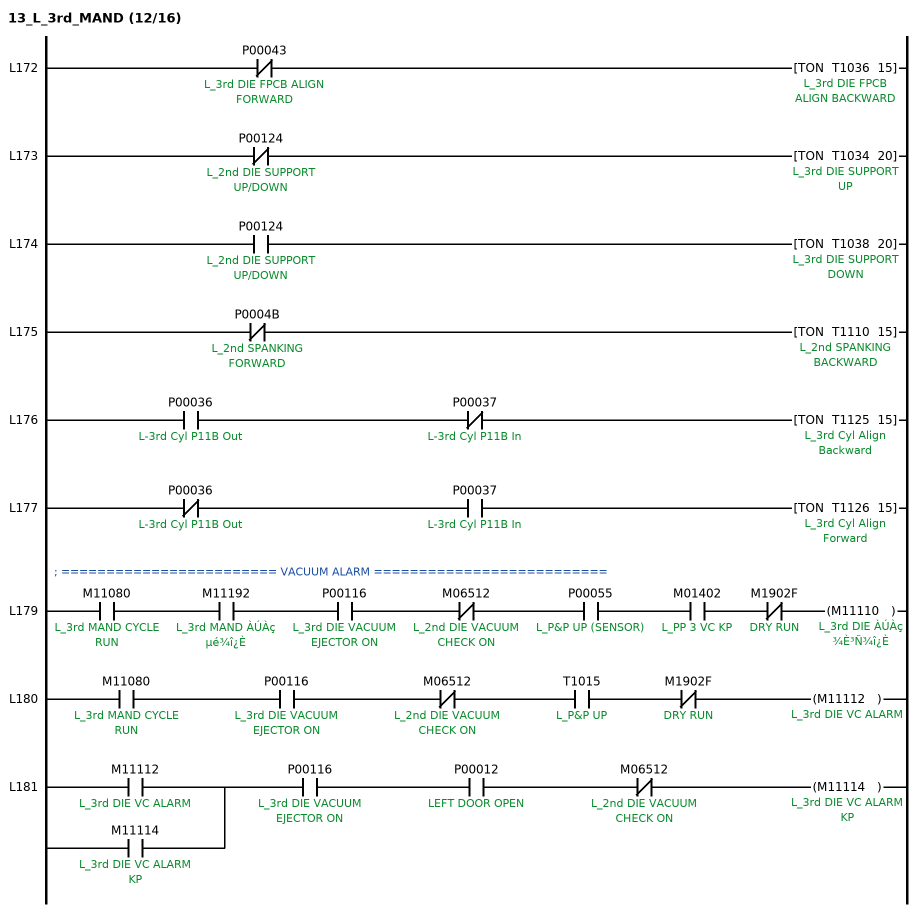
[picture p96: 13_L_3rd_MAND rungs L172-L181]
; L172
LOAD NOT  P00043	// L_3rd DIE FPCB ALIGN FORWARD
TON       T1036 15	// L_3rd DIE FPCB ALIGN BACKWARD
; L173
LOAD NOT  P00124	// L_2nd DIE SUPPORT UP/DOWN
TON       T1034 20	// L_3rd DIE SUPPORT UP
; L174
LOAD      P00124	// L_2nd DIE SUPPORT UP/DOWN
TON       T1038 20	// L_3rd DIE SUPPORT DOWN
; L175
LOAD NOT  P0004B	// L_2nd SPANKING FORWARD
TON       T1110 15	// L_2nd SPANKING BACKWARD
; L176
LOAD      P00036	// L-3rd Cyl P11B Out
AND NOT   P00037	// L-3rd Cyl P11B In
TON       T1125 15	// L_3rd Cyl Align Backward
; L177
LOAD NOT  P00036	// L-3rd Cyl P11B Out
AND       P00037	// L-3rd Cyl P11B In
TON       T1126 15	// L_3rd Cyl Align Forward
// ======================== VACUUM ALARM ==========================
; L179
LOAD      M11080	// L_3rd MAND CYCLE RUN
AND       M11192	// L_3rd MAND ÀÚÀç µé¾î¿È
AND       P00116	// L_3rd DIE VACUUM EJECTOR ON
AND NOT   M06512	// L_2nd DIE VACUUM CHECK ON
AND       P00055	// L_P&P UP (SENSOR)
AND       M01402	// L_PP 3 VC KP
AND NOT   M1902F	// DRY RUN
OUT       M11110	// L_3rd DIE ÀÚÀç ¾È³Ñ¾î¿È
; L180
LOAD      M11080	// L_3rd MAND CYCLE RUN
AND       P00116	// L_3rd DIE VACUUM EJECTOR ON
AND NOT   M06512	// L_2nd DIE VACUUM CHECK ON
AND       T1015	// L_P&P UP
AND NOT   M1902F	// DRY RUN
OUT       M11112	// L_3rd DIE VC ALARM
; L181
LOAD      M11112	// L_3rd DIE VC ALARM
OR        M11114	// L_3rd DIE VC ALARM KP
AND       P00116	// L_3rd DIE VACUUM EJECTOR ON
AND       P00012	// LEFT DOOR OPEN
AND NOT   M06512	// L_2nd DIE VACUUM CHECK ON
OUT       M11114	// L_3rd DIE VC ALARM KP

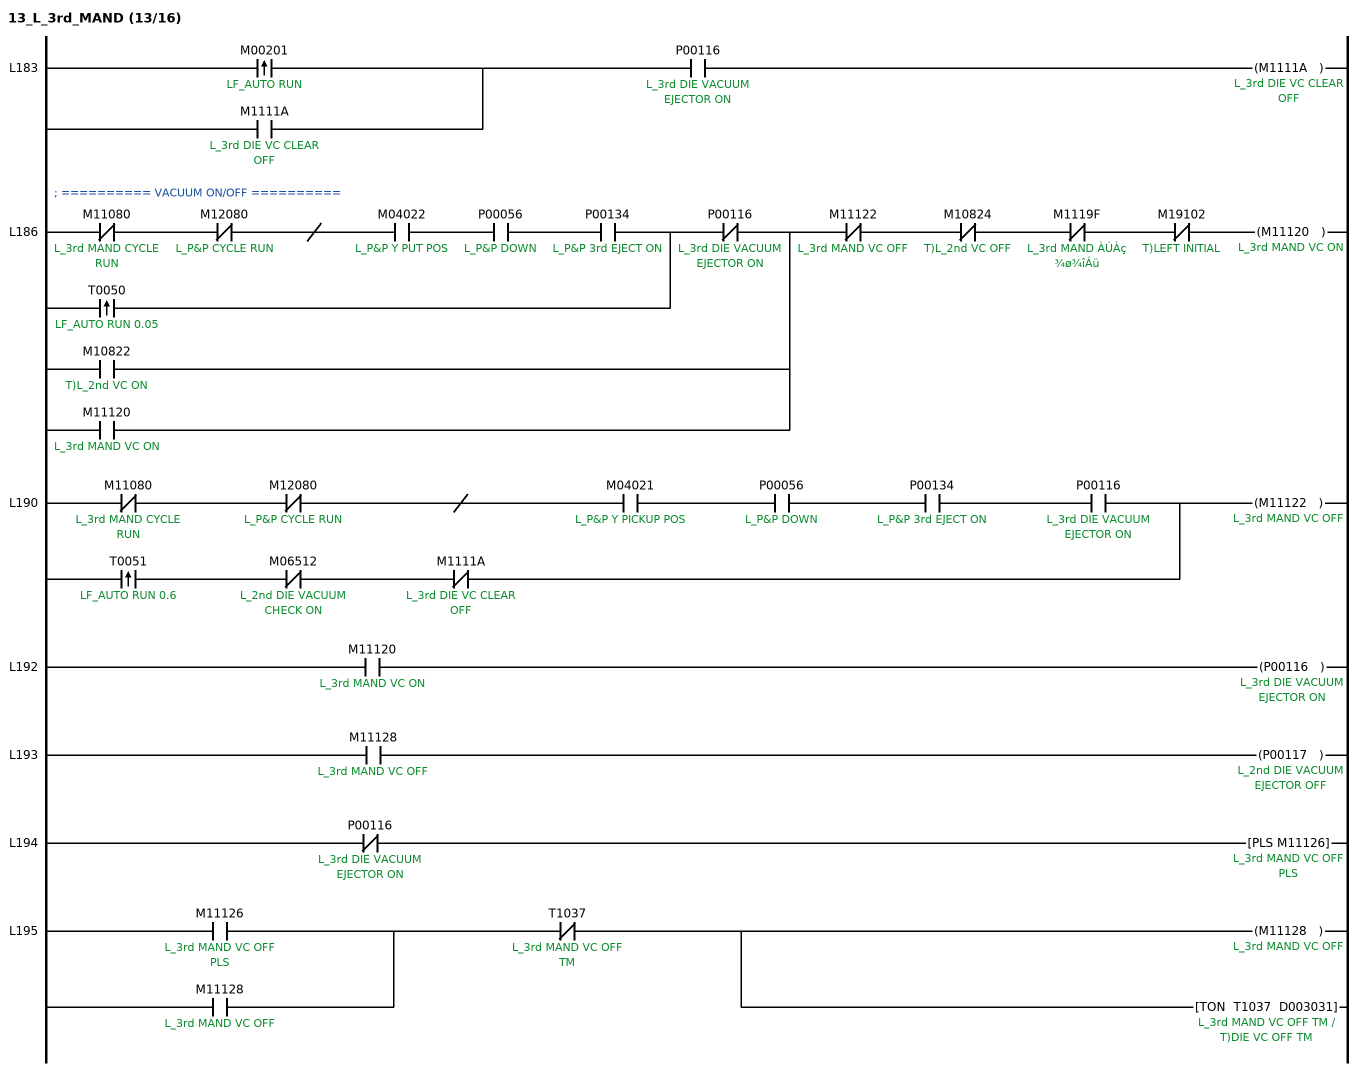
; L183
LOADP     M00201	// LF_AUTO RUN
OR        M1111A	// L_3rd DIE VC CLEAR OFF
AND       P00116	// L_3rd DIE VACUUM EJECTOR ON
OUT       M1111A	// L_3rd DIE VC CLEAR OFF
// ========== VACUUM ON/OFF ==========
; L186
LOAD NOT  M11080	// L_3rd MAND CYCLE RUN
AND NOT   M12080	// L_P&P CYCLE RUN
NOT
AND       M04022	// L_P&P Y PUT POS
AND       P00056	// L_P&P DOWN
AND       P00134	// L_P&P 3rd EJECT ON
ORP       T0050	// LF_AUTO RUN 0.05
AND NOT   P00116	// L_3rd DIE VACUUM EJECTOR ON
OR        M10822	// T)L_2nd VC ON
OR        M11120	// L_3rd MAND VC ON
AND NOT   M11122	// L_3rd MAND VC OFF
AND NOT   M10824	// T)L_2nd VC OFF
AND NOT   M1119F	// L_3rd MAND ÀÚÀç ¾ø¾îÁü
AND NOT   M19102	// T)LEFT INITIAL
OUT       M11120	// L_3rd MAND VC ON
; L190
LOAD NOT  M11080	// L_3rd MAND CYCLE RUN
AND NOT   M12080	// L_P&P CYCLE RUN
NOT
AND       M04021	// L_P&P Y PICKUP POS
AND       P00056	// L_P&P DOWN
AND       P00134	// L_P&P 3rd EJECT ON
AND       P00116	// L_3rd DIE VACUUM EJECTOR ON
LOADP     T0051	// LF_AUTO RUN 0.6
AND NOT   M06512	// L_2nd DIE VACUUM CHECK ON
AND NOT   M1111A	// L_3rd DIE VC CLEAR OFF
OR LOAD
OUT       M11122	// L_3rd MAND VC OFF
; L192
LOAD      M11120	// L_3rd MAND VC ON
OUT       P00116	// L_3rd DIE VACUUM EJECTOR ON
; L193
LOAD      M11128	// L_3rd MAND VC OFF
OUT       P00117	// L_2nd DIE VACUUM EJECTOR OFF
; L194
LOAD NOT  P00116	// L_3rd DIE VACUUM EJECTOR ON
OUTP      M11126	// L_3rd MAND VC OFF PLS
; L195
LOAD      M11126	// L_3rd MAND VC OFF PLS
OR        M11128	// L_3rd MAND VC OFF
AND NOT   T1037	// L_3rd MAND VC OFF TM
OUT       M11128	// L_3rd MAND VC OFF
TON       T1037 D003031	// L_3rd MAND VC OFF TM / T)DIE VC OFF TM

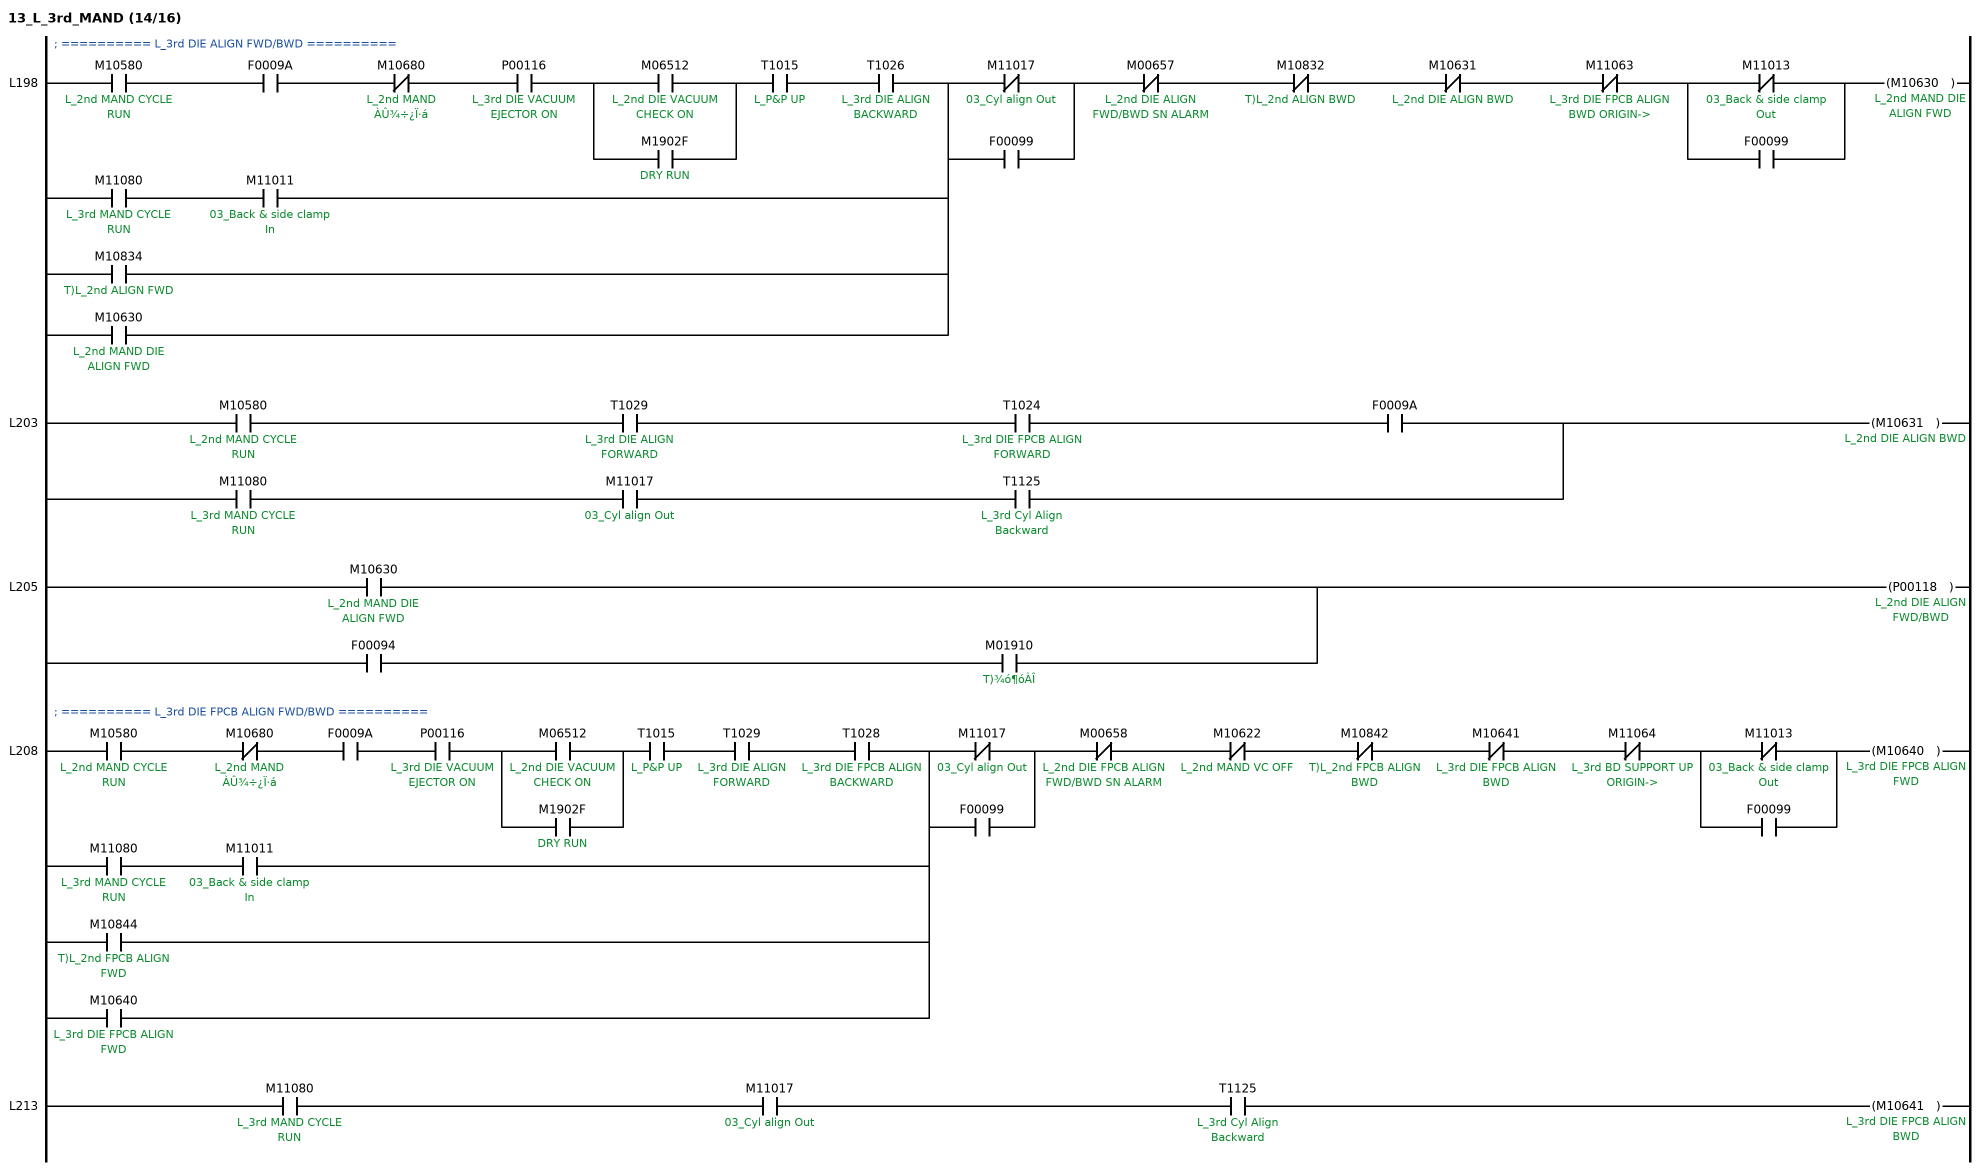
// ========== L_3rd DIE ALIGN FWD/BWD ==========
; L198
LOAD      M10580	// L_2nd MAND CYCLE RUN
AND       F0009A
AND NOT   M10680	// L_2nd MAND ÀÛ¾÷¿Ï·á
AND       P00116	// L_3rd DIE VACUUM EJECTOR ON
LOAD      M06512	// L_2nd DIE VACUUM CHECK ON
OR        M1902F	// DRY RUN
AND LOAD
AND       T1015	// L_P&P UP
AND       T1026	// L_3rd DIE ALIGN BACKWARD
LOAD      M11080	// L_3rd MAND CYCLE RUN
AND       M11011	// 03_Back & side clamp In
OR LOAD
OR        M10834	// T)L_2nd ALIGN FWD
OR        M10630	// L_2nd MAND DIE ALIGN FWD
LOAD NOT  M11017	// 03_Cyl align Out
OR        F00099
AND LOAD
AND NOT   M00657	// L_2nd DIE ALIGN FWD/BWD SN ALARM
AND NOT   M10832	// T)L_2nd ALIGN BWD
AND NOT   M10631	// L_2nd DIE ALIGN BWD
AND NOT   M11063	// L_3rd DIE FPCB ALIGN BWD ORIGIN->
LOAD NOT  M11013	// 03_Back & side clamp Out
OR        F00099
AND LOAD
OUT       M10630	// L_2nd MAND DIE ALIGN FWD
; L203
LOAD      M10580	// L_2nd MAND CYCLE RUN
AND       T1029	// L_3rd DIE ALIGN FORWARD
AND       T1024	// L_3rd DIE FPCB ALIGN FORWARD
AND       F0009A
LOAD      M11080	// L_3rd MAND CYCLE RUN
AND       M11017	// 03_Cyl align Out
AND       T1125	// L_3rd Cyl Align Backward
OR LOAD
OUT       M10631	// L_2nd DIE ALIGN BWD
; L205
LOAD      M10630	// L_2nd MAND DIE ALIGN FWD
LOAD      F00094
AND       M01910	// T)¾ó¶óÀÎ
OR LOAD
OUT       P00118	// L_2nd DIE ALIGN FWD/BWD
// ========== L_3rd DIE FPCB ALIGN FWD/BWD ==========
; L208
LOAD      M10580	// L_2nd MAND CYCLE RUN
AND NOT   M10680	// L_2nd MAND ÀÛ¾÷¿Ï·á
AND       F0009A
AND       P00116	// L_3rd DIE VACUUM EJECTOR ON
LOAD      M06512	// L_2nd DIE VACUUM CHECK ON
OR        M1902F	// DRY RUN
AND LOAD
AND       T1015	// L_P&P UP
AND       T1029	// L_3rd DIE ALIGN FORWARD
AND       T1028	// L_3rd DIE FPCB ALIGN BACKWARD
LOAD      M11080	// L_3rd MAND CYCLE RUN
AND       M11011	// 03_Back & side clamp In
OR LOAD
OR        M10844	// T)L_2nd FPCB ALIGN FWD
OR        M10640	// L_3rd DIE FPCB ALIGN FWD
LOAD NOT  M11017	// 03_Cyl align Out
OR        F00099
AND LOAD
AND NOT   M00658	// L_2nd DIE FPCB ALIGN FWD/BWD SN ALARM
AND NOT   M10622	// L_2nd MAND VC OFF
AND NOT   M10842	// T)L_2nd FPCB ALIGN BWD
AND NOT   M10641	// L_3rd DIE FPCB ALIGN BWD
AND NOT   M11064	// L_3rd BD SUPPORT UP ORIGIN->
LOAD NOT  M11013	// 03_Back & side clamp Out
OR        F00099
AND LOAD
OUT       M10640	// L_3rd DIE FPCB ALIGN FWD
; L213
LOAD      M11080	// L_3rd MAND CYCLE RUN
AND       M11017	// 03_Cyl align Out
AND       T1125	// L_3rd Cyl Align Backward
OUT       M10641	// L_3rd DIE FPCB ALIGN BWD

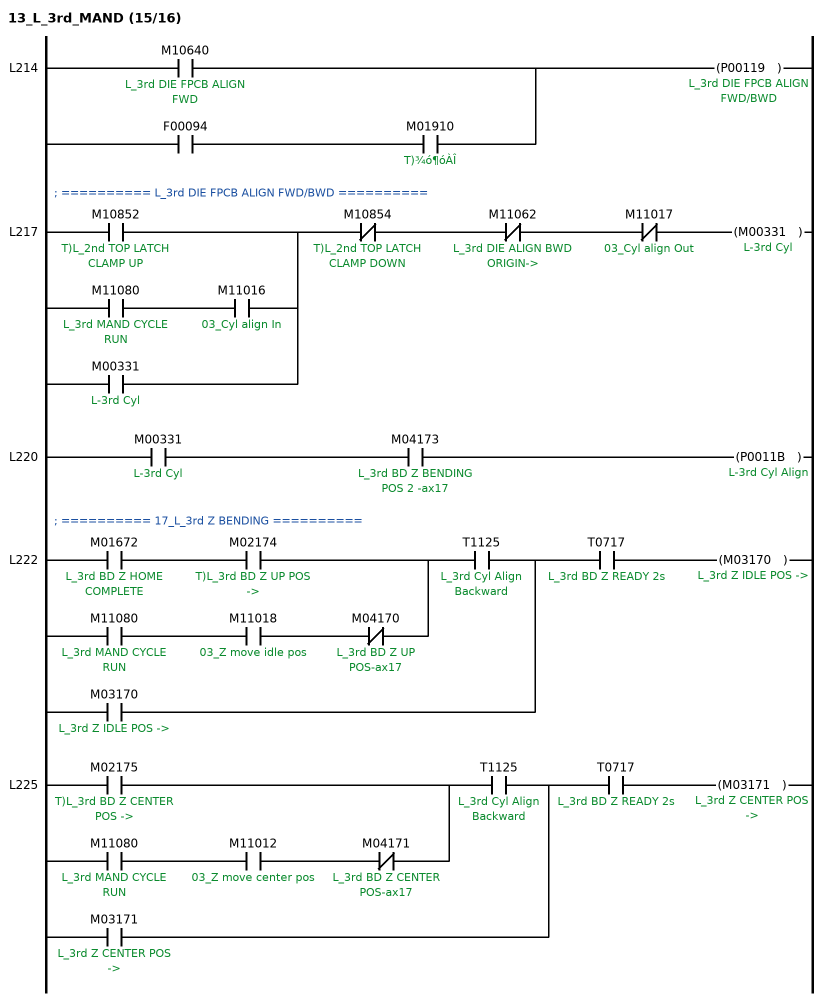
; L214
LOAD      M10640	// L_3rd DIE FPCB ALIGN FWD
LOAD      F00094
AND       M01910	// T)¾ó¶óÀÎ
OR LOAD
OUT       P00119	// L_3rd DIE FPCB ALIGN FWD/BWD
// ========== L_3rd DIE FPCB ALIGN FWD/BWD ==========
; L217
LOAD      M10852	// T)L_2nd TOP LATCH CLAMP UP
LOAD      M11080	// L_3rd MAND CYCLE RUN
AND       M11016	// 03_Cyl align In
OR LOAD
OR        M00331	// L-3rd Cyl
AND NOT   M10854	// T)L_2nd TOP LATCH CLAMP DOWN
AND NOT   M11062	// L_3rd DIE ALIGN BWD ORIGIN->
AND NOT   M11017	// 03_Cyl align Out
OUT       M00331	// L-3rd Cyl
; L220
LOAD      M00331	// L-3rd Cyl
AND       M04173	// L_3rd BD Z BENDING POS 2 -ax17
OUT       P0011B	// L-3rd Cyl Align
// ========== 17_L_3rd Z BENDING ==========
; L222
LOAD      M01672	// L_3rd BD Z HOME COMPLETE
AND       M02174	// T)L_3rd BD Z UP POS ->
LOAD      M11080	// L_3rd MAND CYCLE RUN
AND       M11018	// 03_Z move idle pos
AND NOT   M04170	// L_3rd BD Z UP POS-ax17
OR LOAD
AND       T1125	// L_3rd Cyl Align Backward
OR        M03170	// L_3rd Z IDLE POS ->
AND       T0717	// L_3rd BD Z READY 2s
OUT       M03170	// L_3rd Z IDLE POS ->
; L225
LOAD      M02175	// T)L_3rd BD Z CENTER POS ->
LOAD      M11080	// L_3rd MAND CYCLE RUN
AND       M11012	// 03_Z move center pos
AND NOT   M04171	// L_3rd BD Z CENTER POS-ax17
OR LOAD
AND       T1125	// L_3rd Cyl Align Backward
OR        M03171	// L_3rd Z CENTER POS ->
AND       T0717	// L_3rd BD Z READY 2s
OUT       M03171	// L_3rd Z CENTER POS ->

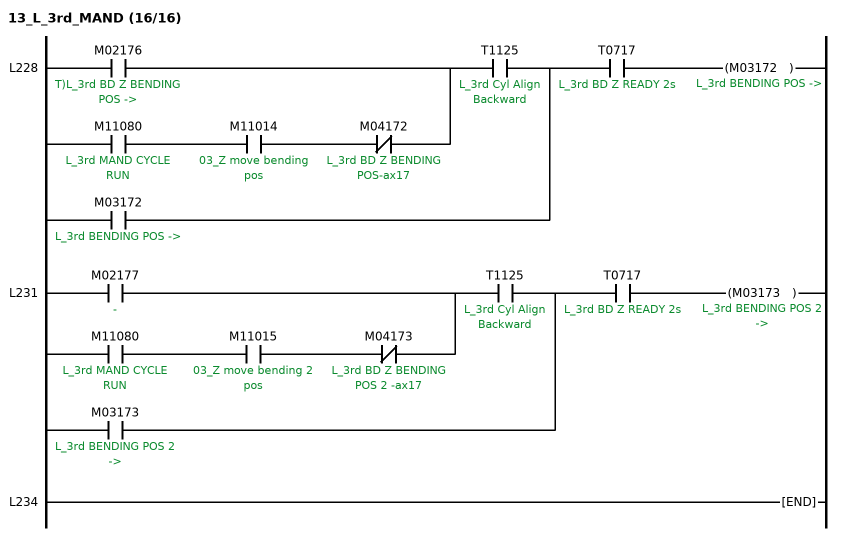
; L228
LOAD      M02176	// T)L_3rd BD Z BENDING POS ->
LOAD      M11080	// L_3rd MAND CYCLE RUN
AND       M11014	// 03_Z move bending pos
AND NOT   M04172	// L_3rd BD Z BENDING POS-ax17
OR LOAD
AND       T1125	// L_3rd Cyl Align Backward
OR        M03172	// L_3rd BENDING POS ->
AND       T0717	// L_3rd BD Z READY 2s
OUT       M03172	// L_3rd BENDING POS ->
; L231
LOAD      M02177	// -
LOAD      M11080	// L_3rd MAND CYCLE RUN
AND       M11015	// 03_Z move bending 2 pos
AND NOT   M04173	// L_3rd BD Z BENDING POS 2 -ax17
OR LOAD
AND       T1125	// L_3rd Cyl Align Backward
OR        M03173	// L_3rd BENDING POS 2 ->
AND       T0717	// L_3rd BD Z READY 2s
OUT       M03173	// L_3rd BENDING POS 2 ->
; L234
END

PROGRAM 14_L_TOOL (task: ½ºÄµ ÇÁ·Î±×·¥)

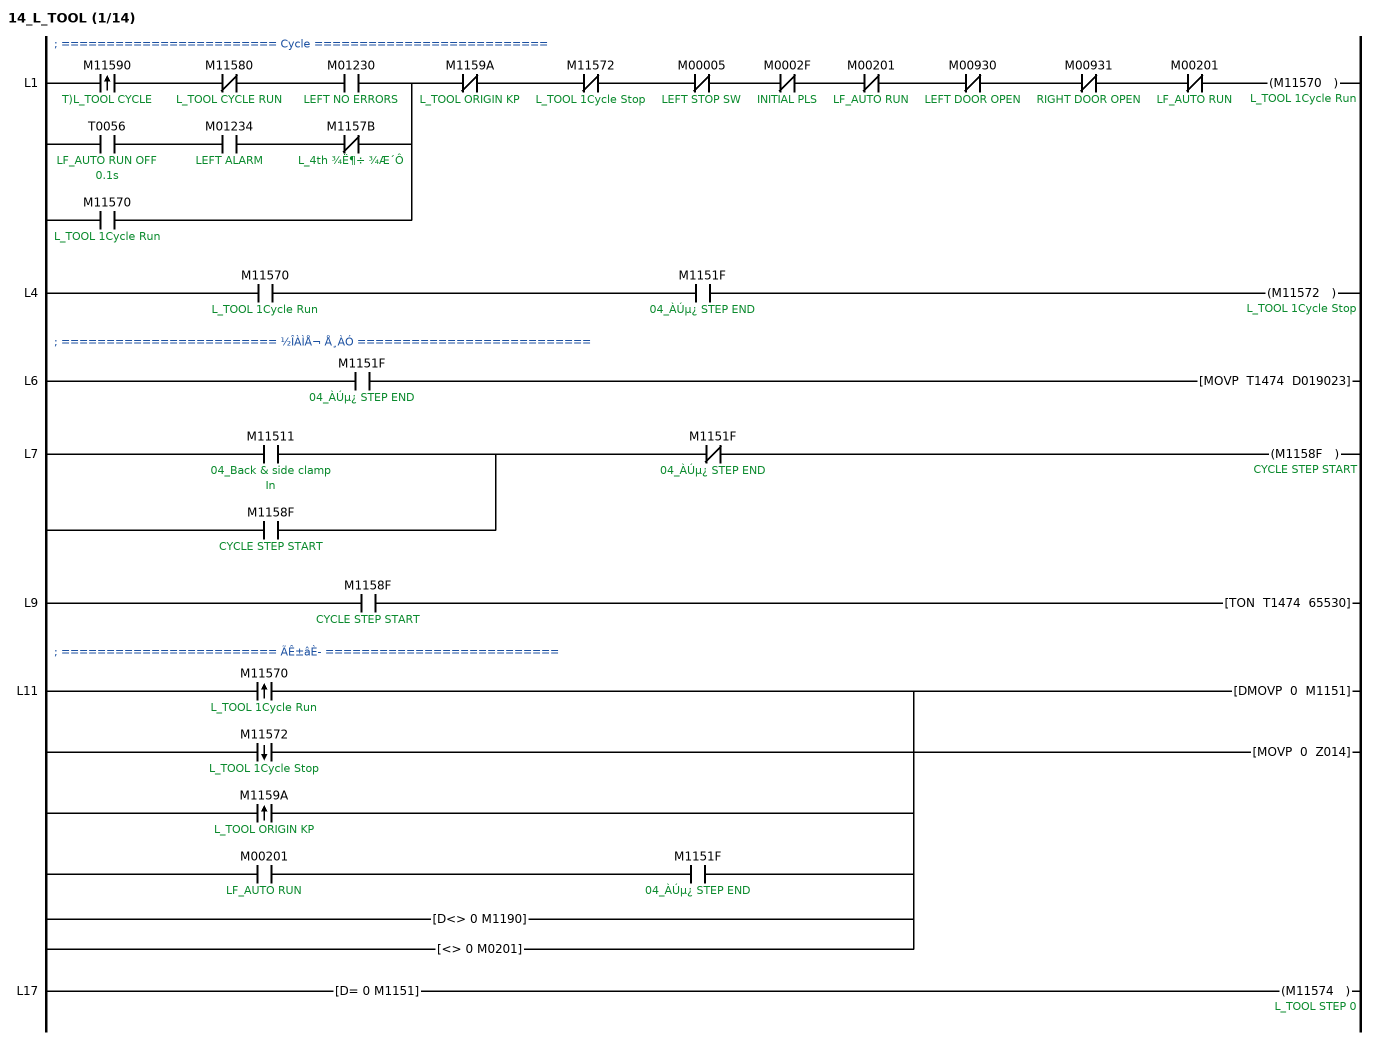
// ======================== Cycle ==========================
; L1
LOADP     M11590	// T)L_TOOL CYCLE
AND NOT   M11580	// L_TOOL CYCLE RUN
AND       M01230	// LEFT NO ERRORS
LOAD      T0056	// LF_AUTO RUN OFF 0.1s
AND       M01234	// LEFT ALARM
AND NOT   M1157B	// L_4th ¾Ë¶÷ ¾Æ´Ô
OR LOAD
OR        M11570	// L_TOOL 1Cycle Run
AND NOT   M1159A	// L_TOOL ORIGIN KP
AND NOT   M11572	// L_TOOL 1Cycle Stop
AND NOT   M00005	// LEFT STOP SW
AND NOT   M0002F	// INITIAL PLS
AND NOT   M00201	// LF_AUTO RUN
AND NOT   M00930	// LEFT DOOR OPEN
AND NOT   M00931	// RIGHT DOOR OPEN
AND NOT   M00201	// LF_AUTO RUN
OUT       M11570	// L_TOOL 1Cycle Run
; L4
LOAD      M11570	// L_TOOL 1Cycle Run
AND       M1151F	// 04_ÀÚµ¿ STEP END
OUT       M11572	// L_TOOL 1Cycle Stop
// ======================== ½ÎÀÌÅ¬ Å¸ÀÓ ==========================
; L6
LOAD      M1151F	// 04_ÀÚµ¿ STEP END
MOVP      T1474 D019023
; L7
LOAD      M11511	// 04_Back & side clamp In
OR        M1158F	// CYCLE STEP START
AND NOT   M1151F	// 04_ÀÚµ¿ STEP END
OUT       M1158F	// CYCLE STEP START
; L9
LOAD      M1158F	// CYCLE STEP START
TON       T1474 65530
// ======================== ÃÊ±âÈ­ ==========================
; L11
LOADP     M11570	// L_TOOL 1Cycle Run
ORN       M11572	// L_TOOL 1Cycle Stop
ORP       M1159A	// L_TOOL ORIGIN KP
LOAD      M00201	// LF_AUTO RUN
AND       M1151F	// 04_ÀÚµ¿ STEP END
OR LOAD
ORD<>     0 M1190
OR<>      0 M0201
DMOVP     0 M1151
MOVP      0 Z014
; L17
LOADD=    0 M1151
OUT       M11574	// L_TOOL STEP 0

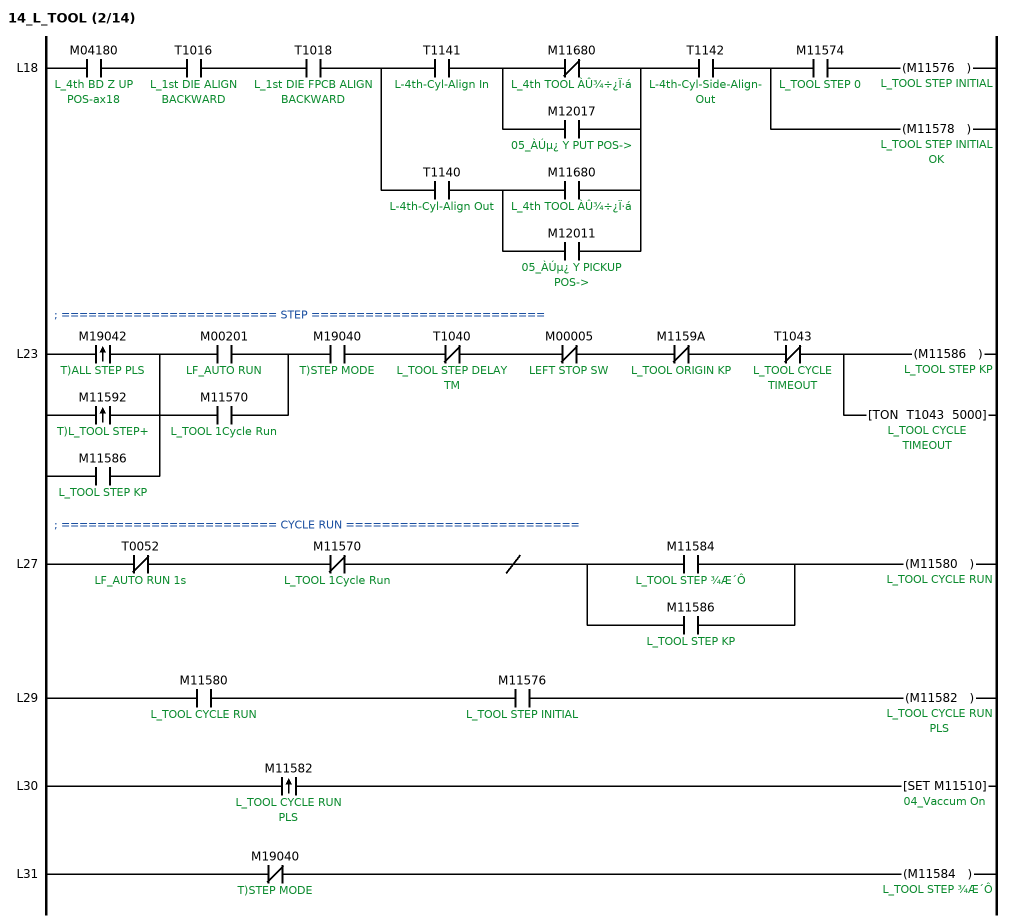
; L18
LOAD      M04180	// L_4th BD Z UP POS-ax18
AND       T1016	// L_1st DIE ALIGN BACKWARD
AND       T1018	// L_1st DIE FPCB ALIGN BACKWARD
LOAD      T1141	// L-4th-Cyl-Align In
LOAD NOT  M11680	// L_4th TOOL ÀÛ¾÷¿Ï·á
OR        M12017	// 05_ÀÚµ¿ Y PUT POS->
AND LOAD
LOAD      T1140	// L-4th-Cyl-Align Out
LOAD      M11680	// L_4th TOOL ÀÛ¾÷¿Ï·á
OR        M12011	// 05_ÀÚµ¿ Y PICKUP POS->
AND LOAD
OR LOAD
AND LOAD
AND       T1142	// L-4th-Cyl-Side-Align-Out
MPUSH
AND       M11574	// L_TOOL STEP 0
OUT       M11576	// L_TOOL STEP INITIAL
MPOP
OUT       M11578	// L_TOOL STEP INITIAL OK
// ======================== STEP ==========================
; L23
LOADP     M19042	// T)ALL STEP PLS
ORP       M11592	// T)L_TOOL STEP+
OR        M11586	// L_TOOL STEP KP
LOAD      M00201	// LF_AUTO RUN
OR        M11570	// L_TOOL 1Cycle Run
AND LOAD
AND       M19040	// T)STEP MODE
AND NOT   T1040	// L_TOOL STEP DELAY TM
AND NOT   M00005	// LEFT STOP SW
AND NOT   M1159A	// L_TOOL ORIGIN KP
AND NOT   T1043	// L_TOOL CYCLE TIMEOUT
OUT       M11586	// L_TOOL STEP KP
TON       T1043 5000	// L_TOOL CYCLE TIMEOUT
// ======================== CYCLE RUN ==========================
; L27
LOAD NOT  T0052	// LF_AUTO RUN 1s
AND NOT   M11570	// L_TOOL 1Cycle Run
NOT
LOAD      M11584	// L_TOOL STEP ¾Æ´Ô
OR        M11586	// L_TOOL STEP KP
AND LOAD
OUT       M11580	// L_TOOL CYCLE RUN
; L29
LOAD      M11580	// L_TOOL CYCLE RUN
AND       M11576	// L_TOOL STEP INITIAL
OUT       M11582	// L_TOOL CYCLE RUN PLS
; L30
LOADP     M11582	// L_TOOL CYCLE RUN PLS
SET       M11510	// 04_Vaccum On
; L31
LOAD NOT  M19040	// T)STEP MODE
OUT       M11584	// L_TOOL STEP ¾Æ´Ô

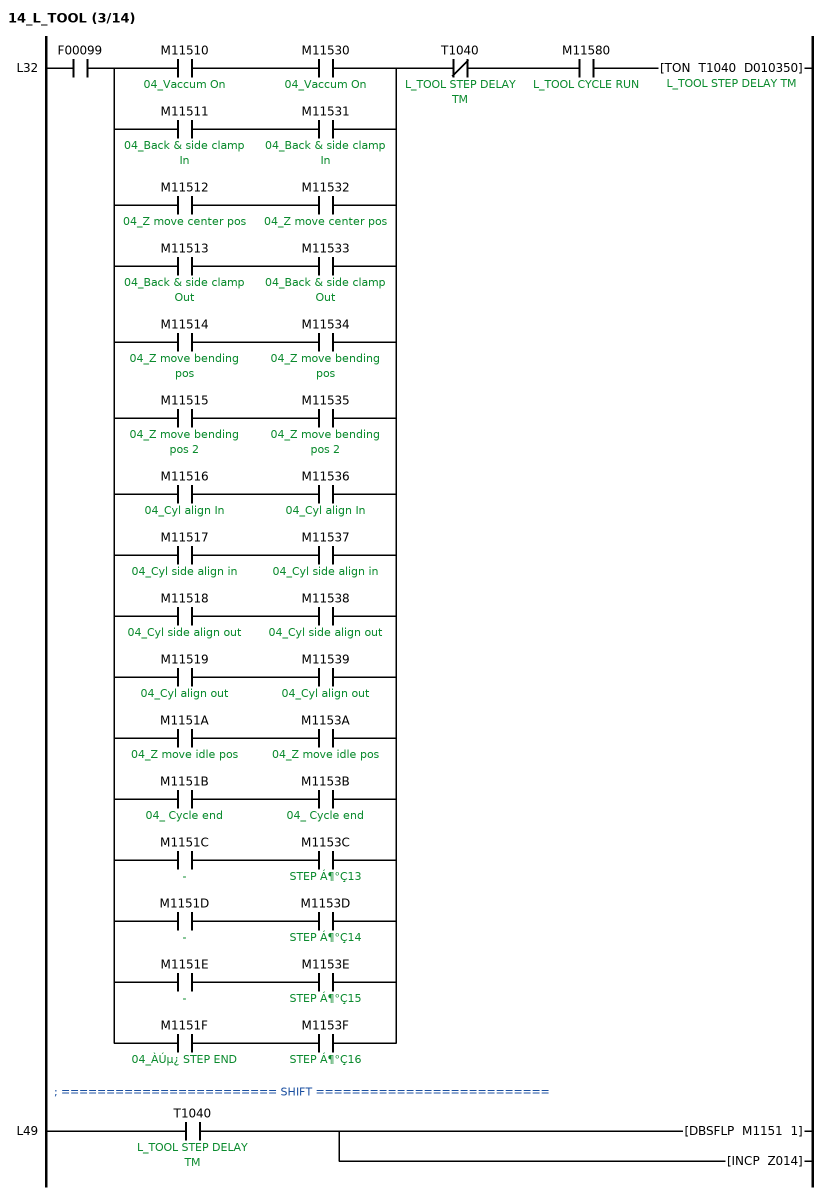
; L32
LOAD      F00099
LOAD      M11510	// 04_Vaccum On
AND       M11530	// 04_Vaccum On
LOAD      M11511	// 04_Back & side clamp In
AND       M11531	// 04_Back & side clamp In
OR LOAD
LOAD      M11512	// 04_Z move center pos
AND       M11532	// 04_Z move center pos
OR LOAD
LOAD      M11513	// 04_Back & side clamp Out
AND       M11533	// 04_Back & side clamp Out
OR LOAD
LOAD      M11514	// 04_Z move bending pos
AND       M11534	// 04_Z move bending pos
OR LOAD
LOAD      M11515	// 04_Z move bending pos 2
AND       M11535	// 04_Z move bending pos 2
OR LOAD
LOAD      M11516	// 04_Cyl align In
AND       M11536	// 04_Cyl align In
OR LOAD
LOAD      M11517	// 04_Cyl side align in
AND       M11537	// 04_Cyl side align in
OR LOAD
LOAD      M11518	// 04_Cyl side align out
AND       M11538	// 04_Cyl side align out
OR LOAD
LOAD      M11519	// 04_Cyl align out
AND       M11539	// 04_Cyl align out
OR LOAD
LOAD      M1151A	// 04_Z move idle pos
AND       M1153A	// 04_Z move idle pos
OR LOAD
LOAD      M1151B	// 04_ Cycle end
AND       M1153B	// 04_ Cycle end
OR LOAD
LOAD      M1151C	// -
AND       M1153C	// STEP Á¶°Ç13
OR LOAD
LOAD      M1151D	// -
AND       M1153D	// STEP Á¶°Ç14
OR LOAD
LOAD      M1151E	// -
AND       M1153E	// STEP Á¶°Ç15
OR LOAD
LOAD      M1151F	// 04_ÀÚµ¿ STEP END
AND       M1153F	// STEP Á¶°Ç16
OR LOAD
AND LOAD
AND NOT   T1040	// L_TOOL STEP DELAY TM
AND       M11580	// L_TOOL CYCLE RUN
TON       T1040 D010350	// L_TOOL STEP DELAY TM
// ======================== SHIFT ==========================
; L49
LOAD      T1040	// L_TOOL STEP DELAY TM
DBSFLP    M1151 1
INCP      Z014

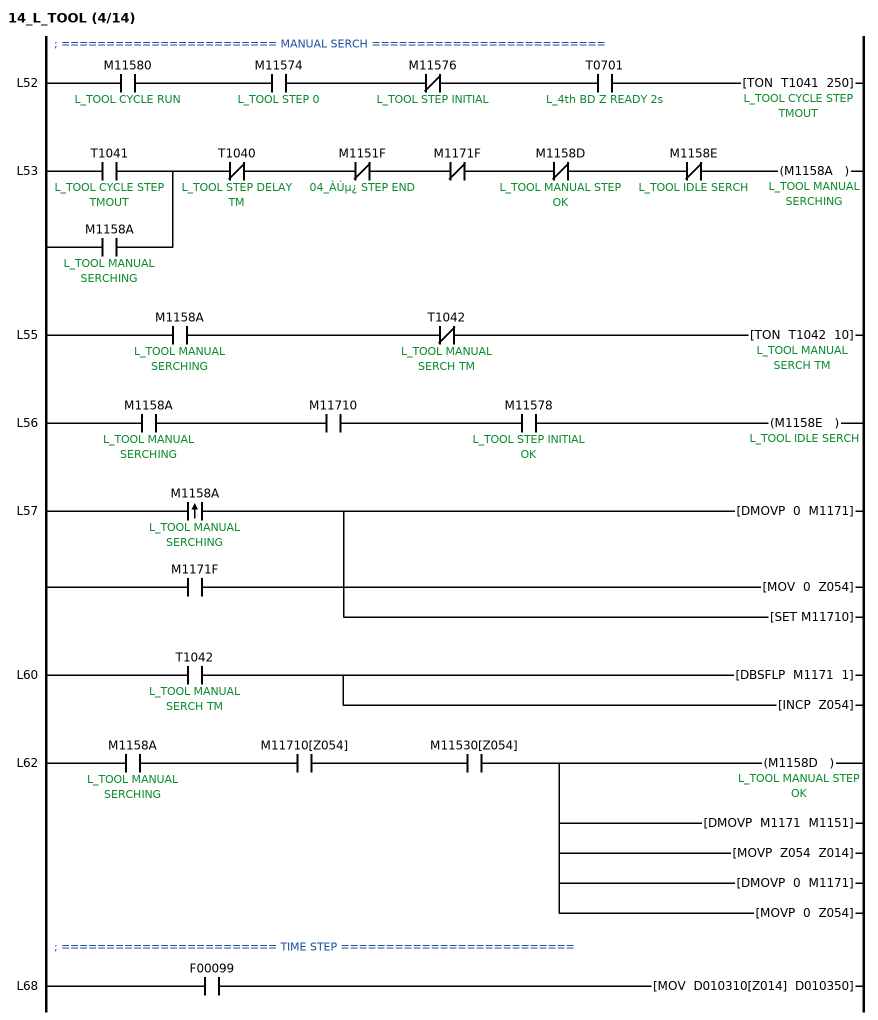
// ======================== MANUAL SERCH ==========================
; L52
LOAD      M11580	// L_TOOL CYCLE RUN
AND       M11574	// L_TOOL STEP 0
AND NOT   M11576	// L_TOOL STEP INITIAL
AND       T0701	// L_4th BD Z READY 2s
TON       T1041 250	// L_TOOL CYCLE STEP TMOUT
; L53
LOAD      T1041	// L_TOOL CYCLE STEP TMOUT
OR        M1158A	// L_TOOL MANUAL SERCHING
AND NOT   T1040	// L_TOOL STEP DELAY TM
AND NOT   M1151F	// 04_ÀÚµ¿ STEP END
AND NOT   M1171F
AND NOT   M1158D	// L_TOOL MANUAL STEP OK
AND NOT   M1158E	// L_TOOL IDLE SERCH
OUT       M1158A	// L_TOOL MANUAL SERCHING
; L55
LOAD      M1158A	// L_TOOL MANUAL SERCHING
AND NOT   T1042	// L_TOOL MANUAL SERCH TM
TON       T1042 10	// L_TOOL MANUAL SERCH TM
; L56
LOAD      M1158A	// L_TOOL MANUAL SERCHING
AND       M11710
AND       M11578	// L_TOOL STEP INITIAL OK
OUT       M1158E	// L_TOOL IDLE SERCH
; L57
LOADP     M1158A	// L_TOOL MANUAL SERCHING
OR        M1171F
DMOVP     0 M1171
MOV       0 Z054
SET       M11710
; L60
LOAD      T1042	// L_TOOL MANUAL SERCH TM
DBSFLP    M1171 1
INCP      Z054
; L62
LOAD      M1158A	// L_TOOL MANUAL SERCHING
AND       M11710[Z054]
AND       M11530[Z054]
OUT       M1158D	// L_TOOL MANUAL STEP OK
DMOVP     M1171 M1151
MOVP      Z054 Z014
DMOVP     0 M1171
MOVP      0 Z054
// ======================== TIME STEP ==========================
; L68
LOAD      F00099
MOV       D010310[Z014] D010350

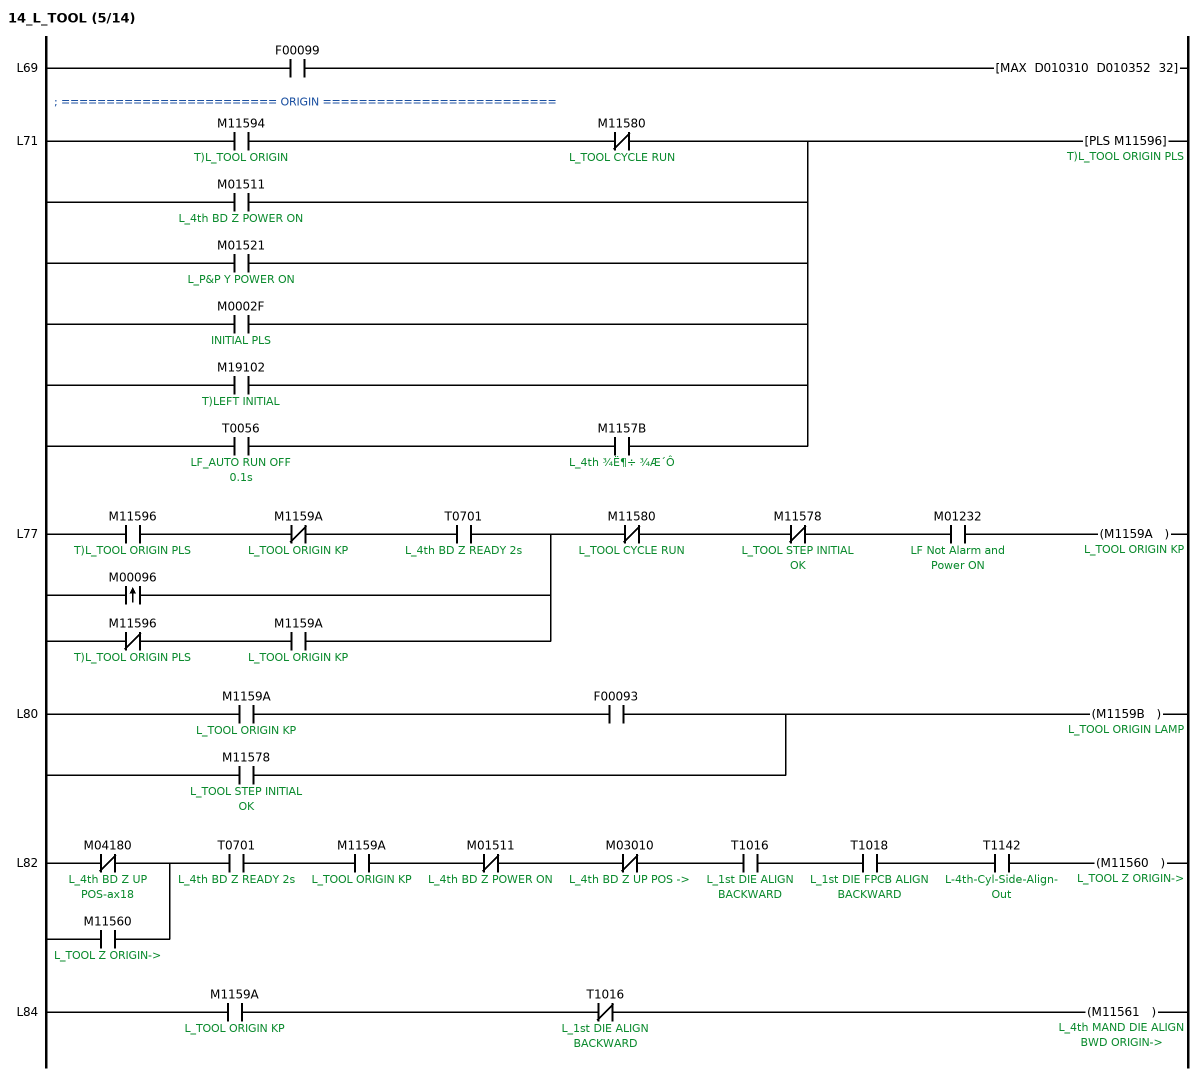
; L69
LOAD      F00099
MAX       D010310 D010352 32
// ======================== ORIGIN ==========================
; L71
LOAD      M11594	// T)L_TOOL ORIGIN
AND NOT   M11580	// L_TOOL CYCLE RUN
OR        M01511	// L_4th BD Z POWER ON
OR        M01521	// L_P&P Y POWER ON
OR        M0002F	// INITIAL PLS
OR        M19102	// T)LEFT INITIAL
LOAD      T0056	// LF_AUTO RUN OFF 0.1s
AND       M1157B	// L_4th ¾Ë¶÷ ¾Æ´Ô
OR LOAD
OUTP      M11596	// T)L_TOOL ORIGIN PLS
; L77
LOAD      M11596	// T)L_TOOL ORIGIN PLS
AND NOT   M1159A	// L_TOOL ORIGIN KP
AND       T0701	// L_4th BD Z READY 2s
ORP       M00096
LOAD NOT  M11596	// T)L_TOOL ORIGIN PLS
AND       M1159A	// L_TOOL ORIGIN KP
OR LOAD
AND NOT   M11580	// L_TOOL CYCLE RUN
AND NOT   M11578	// L_TOOL STEP INITIAL OK
AND       M01232	// LF Not Alarm and Power ON
OUT       M1159A	// L_TOOL ORIGIN KP
; L80
LOAD      M1159A	// L_TOOL ORIGIN KP
AND       F00093
OR        M11578	// L_TOOL STEP INITIAL OK
OUT       M1159B	// L_TOOL ORIGIN LAMP
; L82
LOAD NOT  M04180	// L_4th BD Z UP POS-ax18
OR        M11560	// L_TOOL Z ORIGIN->
AND       T0701	// L_4th BD Z READY 2s
AND       M1159A	// L_TOOL ORIGIN KP
AND NOT   M01511	// L_4th BD Z POWER ON
AND NOT   M03010	// L_4th BD Z UP POS ->
AND       T1016	// L_1st DIE ALIGN BACKWARD
AND       T1018	// L_1st DIE FPCB ALIGN BACKWARD
AND       T1142	// L-4th-Cyl-Side-Align-Out
OUT       M11560	// L_TOOL Z ORIGIN->
; L84
LOAD      M1159A	// L_TOOL ORIGIN KP
AND NOT   T1016	// L_1st DIE ALIGN BACKWARD
OUT       M11561	// L_4th MAND DIE ALIGN BWD ORIGIN->

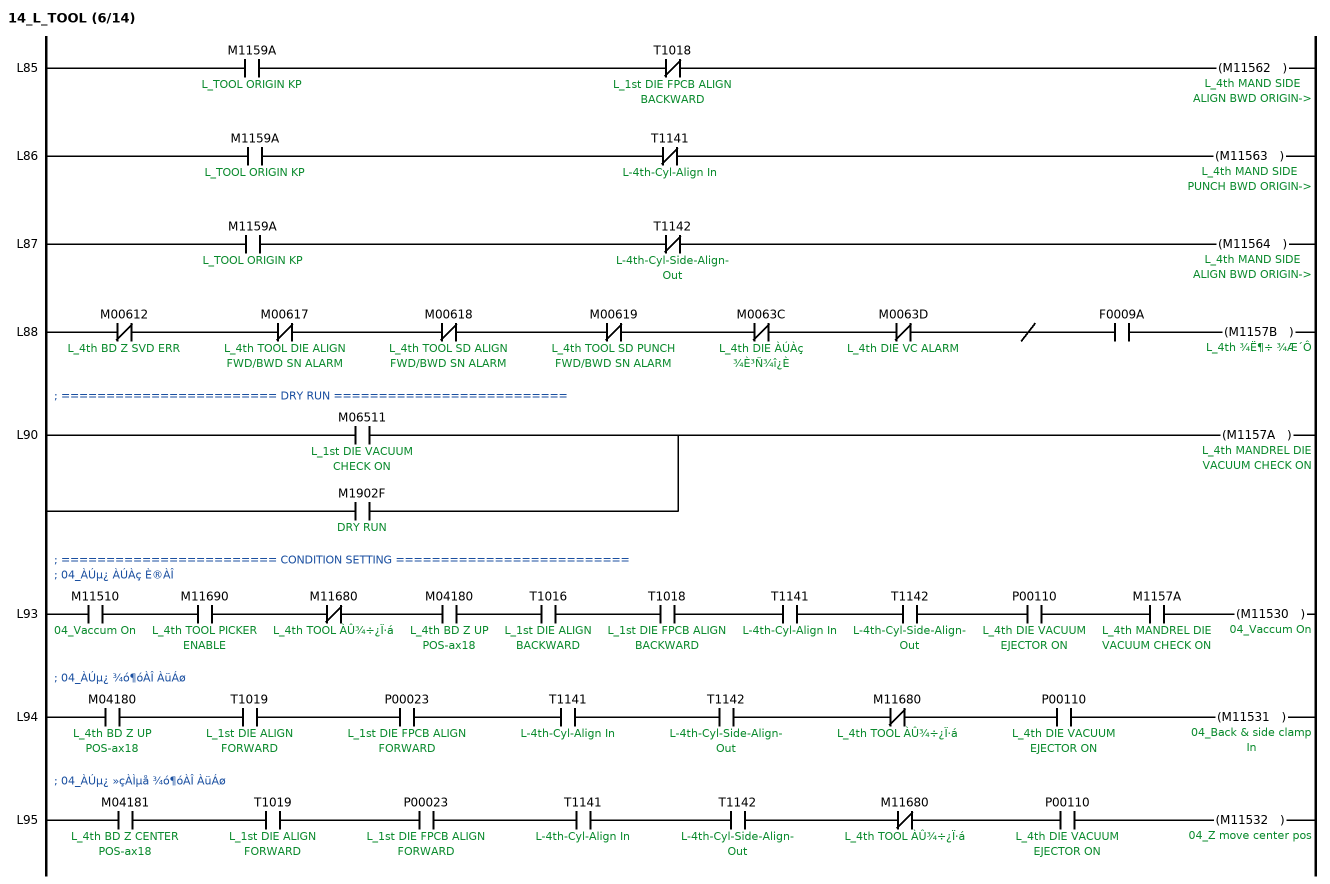
; L85
LOAD      M1159A	// L_TOOL ORIGIN KP
AND NOT   T1018	// L_1st DIE FPCB ALIGN BACKWARD
OUT       M11562	// L_4th MAND SIDE ALIGN BWD ORIGIN->
; L86
LOAD      M1159A	// L_TOOL ORIGIN KP
AND NOT   T1141	// L-4th-Cyl-Align In
OUT       M11563	// L_4th MAND SIDE PUNCH BWD ORIGIN->
; L87
LOAD      M1159A	// L_TOOL ORIGIN KP
AND NOT   T1142	// L-4th-Cyl-Side-Align-Out
OUT       M11564	// L_4th MAND SIDE ALIGN BWD ORIGIN->
; L88
LOAD NOT  M00612	// L_4th BD Z SVD ERR
AND NOT   M00617	// L_4th TOOL DIE ALIGN FWD/BWD SN ALARM
AND NOT   M00618	// L_4th TOOL SD ALIGN FWD/BWD SN ALARM
AND NOT   M00619	// L_4th TOOL SD PUNCH FWD/BWD SN ALARM
AND NOT   M0063C	// L_4th DIE ÀÚÀç ¾È³Ñ¾î¿È
AND NOT   M0063D	// L_4th DIE VC ALARM
NOT
AND       F0009A
OUT       M1157B	// L_4th ¾Ë¶÷ ¾Æ´Ô
// ======================== DRY RUN ==========================
; L90
LOAD      M06511	// L_1st DIE VACUUM CHECK ON
OR        M1902F	// DRY RUN
OUT       M1157A	// L_4th MANDREL DIE VACUUM CHECK ON
// ======================== CONDITION SETTING ==========================
; L93
LOAD      M11510	// 04_Vaccum On
AND       M11690	// L_4th TOOL PICKER ENABLE
AND NOT   M11680	// L_4th TOOL ÀÛ¾÷¿Ï·á
AND       M04180	// L_4th BD Z UP POS-ax18
AND       T1016	// L_1st DIE ALIGN BACKWARD
AND       T1018	// L_1st DIE FPCB ALIGN BACKWARD
AND       T1141	// L-4th-Cyl-Align In
AND       T1142	// L-4th-Cyl-Side-Align-Out
AND       P00110	// L_4th DIE VACUUM EJECTOR ON
AND       M1157A	// L_4th MANDREL DIE VACUUM CHECK ON
OUT       M11530	// 04_Vaccum On
// output comment: 04_ÀÚµ¿ ÀÚÀç È®ÀÎ
; L94
LOAD      M04180	// L_4th BD Z UP POS-ax18
AND       T1019	// L_1st DIE ALIGN FORWARD
AND       P00023	// L_1st DIE FPCB ALIGN FORWARD
AND       T1141	// L-4th-Cyl-Align In
AND       T1142	// L-4th-Cyl-Side-Align-Out
AND NOT   M11680	// L_4th TOOL ÀÛ¾÷¿Ï·á
AND       P00110	// L_4th DIE VACUUM EJECTOR ON
OUT       M11531	// 04_Back & side clamp In
// output comment: 04_ÀÚµ¿ ¾ó¶óÀÎ ÀüÁø
; L95
LOAD      M04181	// L_4th BD Z CENTER POS-ax18
AND       T1019	// L_1st DIE ALIGN FORWARD
AND       P00023	// L_1st DIE FPCB ALIGN FORWARD
AND       T1141	// L-4th-Cyl-Align In
AND       T1142	// L-4th-Cyl-Side-Align-Out
AND NOT   M11680	// L_4th TOOL ÀÛ¾÷¿Ï·á
AND       P00110	// L_4th DIE VACUUM EJECTOR ON
OUT       M11532	// 04_Z move center pos
// output comment: 04_ÀÚµ¿ »çÀÌµå ¾ó¶óÀÎ ÀüÁø

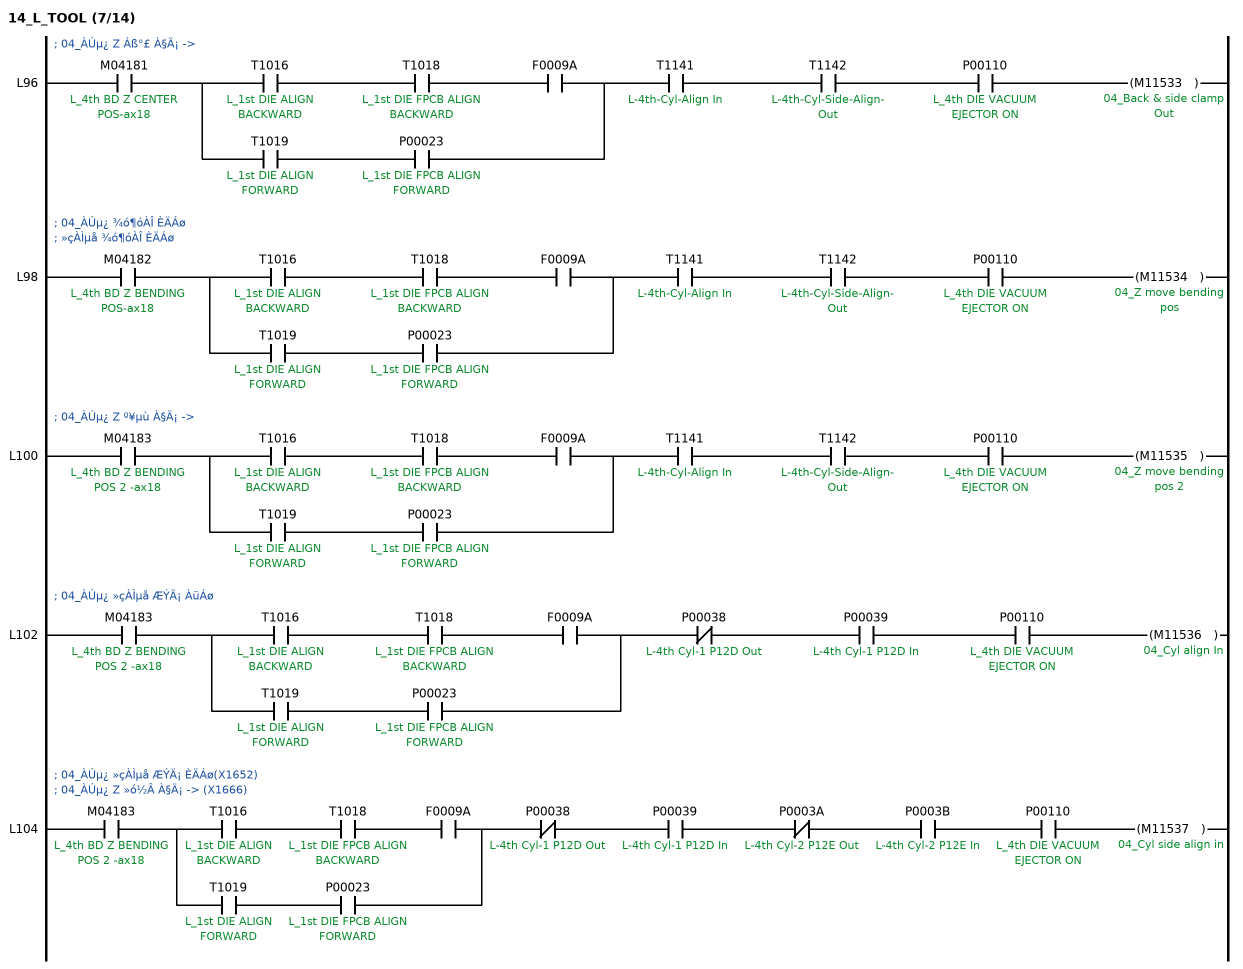
; L96
LOAD      M04181	// L_4th BD Z CENTER POS-ax18
LOAD      T1016	// L_1st DIE ALIGN BACKWARD
AND       T1018	// L_1st DIE FPCB ALIGN BACKWARD
AND       F0009A
LOAD      T1019	// L_1st DIE ALIGN FORWARD
AND       P00023	// L_1st DIE FPCB ALIGN FORWARD
OR LOAD
AND LOAD
AND       T1141	// L-4th-Cyl-Align In
AND       T1142	// L-4th-Cyl-Side-Align-Out
AND       P00110	// L_4th DIE VACUUM EJECTOR ON
OUT       M11533	// 04_Back & side clamp Out
// output comment: 04_ÀÚµ¿ Z Áß°£ À§Ä¡ ->
; L98
LOAD      M04182	// L_4th BD Z BENDING POS-ax18
LOAD      T1016	// L_1st DIE ALIGN BACKWARD
AND       T1018	// L_1st DIE FPCB ALIGN BACKWARD
AND       F0009A
LOAD      T1019	// L_1st DIE ALIGN FORWARD
AND       P00023	// L_1st DIE FPCB ALIGN FORWARD
OR LOAD
AND LOAD
AND       T1141	// L-4th-Cyl-Align In
AND       T1142	// L-4th-Cyl-Side-Align-Out
AND       P00110	// L_4th DIE VACUUM EJECTOR ON
OUT       M11534	// 04_Z move bending pos
// output comment: 04_ÀÚµ¿ ¾ó¶óÀÎ ÈÄÁø »çÀÌµå ¾ó¶óÀÎ ÈÄÁø
; L100
LOAD      M04183	// L_4th BD Z BENDING POS 2 -ax18
LOAD      T1016	// L_1st DIE ALIGN BACKWARD
AND       T1018	// L_1st DIE FPCB ALIGN BACKWARD
AND       F0009A
LOAD      T1019	// L_1st DIE ALIGN FORWARD
AND       P00023	// L_1st DIE FPCB ALIGN FORWARD
OR LOAD
AND LOAD
AND       T1141	// L-4th-Cyl-Align In
AND       T1142	// L-4th-Cyl-Side-Align-Out
AND       P00110	// L_4th DIE VACUUM EJECTOR ON
OUT       M11535	// 04_Z move bending pos 2
// output comment: 04_ÀÚµ¿ Z º¥µù À§Ä¡ ->
; L102
LOAD      M04183	// L_4th BD Z BENDING POS 2 -ax18
LOAD      T1016	// L_1st DIE ALIGN BACKWARD
AND       T1018	// L_1st DIE FPCB ALIGN BACKWARD
AND       F0009A
LOAD      T1019	// L_1st DIE ALIGN FORWARD
AND       P00023	// L_1st DIE FPCB ALIGN FORWARD
OR LOAD
AND LOAD
AND NOT   P00038	// L-4th Cyl-1 P12D Out
AND       P00039	// L-4th Cyl-1 P12D In
AND       P00110	// L_4th DIE VACUUM EJECTOR ON
OUT       M11536	// 04_Cyl align In
// output comment: 04_ÀÚµ¿ »çÀÌµå ÆÝÄ¡ ÀüÁø
; L104
LOAD      M04183	// L_4th BD Z BENDING POS 2 -ax18
LOAD      T1016	// L_1st DIE ALIGN BACKWARD
AND       T1018	// L_1st DIE FPCB ALIGN BACKWARD
AND       F0009A
LOAD      T1019	// L_1st DIE ALIGN FORWARD
AND       P00023	// L_1st DIE FPCB ALIGN FORWARD
OR LOAD
AND LOAD
AND NOT   P00038	// L-4th Cyl-1 P12D Out
AND       P00039	// L-4th Cyl-1 P12D In
AND NOT   P0003A	// L-4th Cyl-2 P12E Out
AND       P0003B	// L-4th Cyl-2 P12E In
AND       P00110	// L_4th DIE VACUUM EJECTOR ON
OUT       M11537	// 04_Cyl side align in
// output comment: 04_ÀÚµ¿ »çÀÌµå ÆÝÄ¡ ÈÄÁø(X1652) 04_ÀÚµ¿ Z »ó½Â À§Ä¡ -> (X1666)

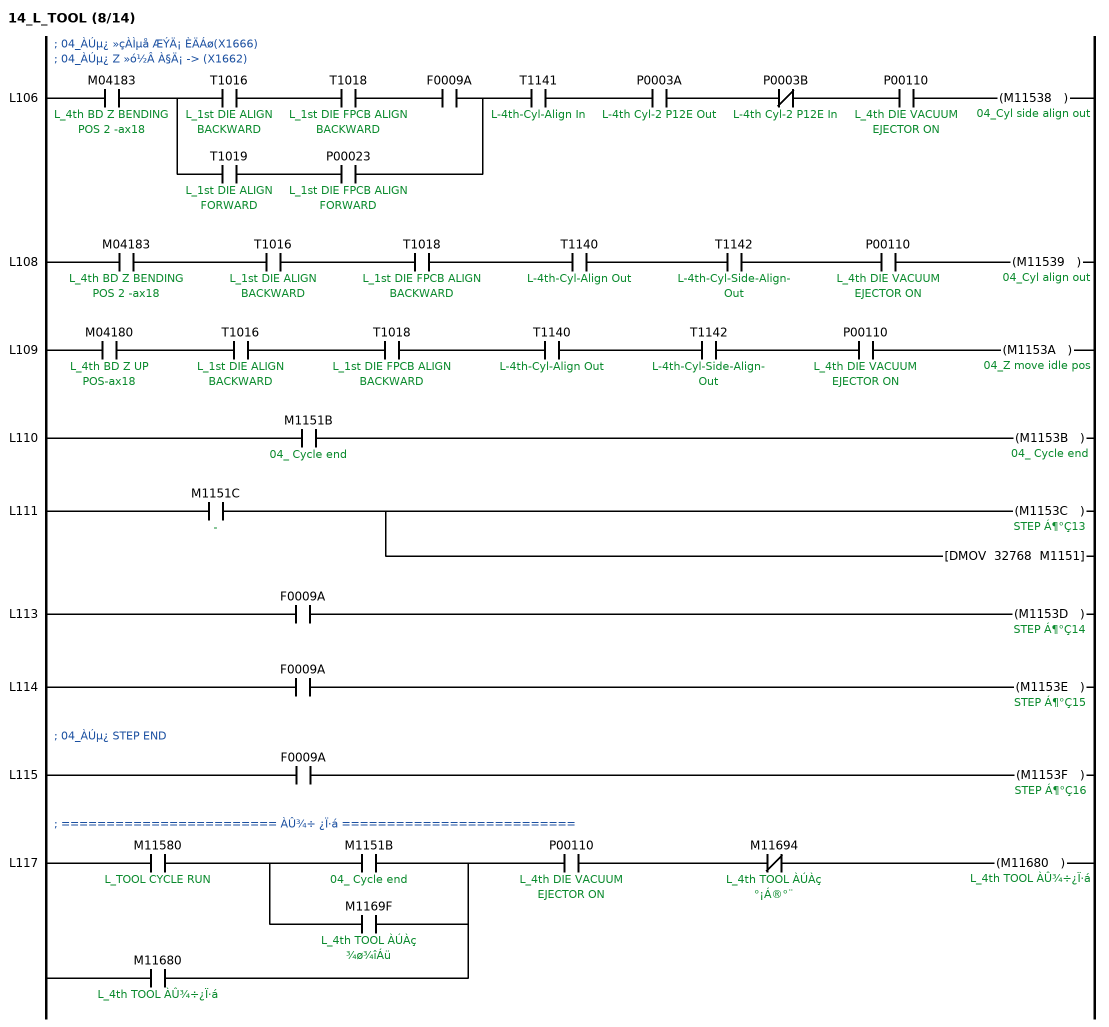
; L106
LOAD      M04183	// L_4th BD Z BENDING POS 2 -ax18
LOAD      T1016	// L_1st DIE ALIGN BACKWARD
AND       T1018	// L_1st DIE FPCB ALIGN BACKWARD
AND       F0009A
LOAD      T1019	// L_1st DIE ALIGN FORWARD
AND       P00023	// L_1st DIE FPCB ALIGN FORWARD
OR LOAD
AND LOAD
AND       T1141	// L-4th-Cyl-Align In
AND       P0003A	// L-4th Cyl-2 P12E Out
AND NOT   P0003B	// L-4th Cyl-2 P12E In
AND       P00110	// L_4th DIE VACUUM EJECTOR ON
OUT       M11538	// 04_Cyl side align out
// output comment: 04_ÀÚµ¿ »çÀÌµå ÆÝÄ¡ ÈÄÁø(X1666) 04_ÀÚµ¿ Z »ó½Â À§Ä¡ -> (X1662)
; L108
LOAD      M04183	// L_4th BD Z BENDING POS 2 -ax18
AND       T1016	// L_1st DIE ALIGN BACKWARD
AND       T1018	// L_1st DIE FPCB ALIGN BACKWARD
AND       T1140	// L-4th-Cyl-Align Out
AND       T1142	// L-4th-Cyl-Side-Align-Out
AND       P00110	// L_4th DIE VACUUM EJECTOR ON
OUT       M11539	// 04_Cyl align out
; L109
LOAD      M04180	// L_4th BD Z UP POS-ax18
AND       T1016	// L_1st DIE ALIGN BACKWARD
AND       T1018	// L_1st DIE FPCB ALIGN BACKWARD
AND       T1140	// L-4th-Cyl-Align Out
AND       T1142	// L-4th-Cyl-Side-Align-Out
AND       P00110	// L_4th DIE VACUUM EJECTOR ON
OUT       M1153A	// 04_Z move idle pos
; L110
LOAD      M1151B	// 04_ Cycle end
OUT       M1153B	// 04_ Cycle end
; L111
LOAD      M1151C	// -
OUT       M1153C	// STEP Á¶°Ç13
DMOV      32768 M1151
; L113
LOAD      F0009A
OUT       M1153D	// STEP Á¶°Ç14
; L114
LOAD      F0009A
OUT       M1153E	// STEP Á¶°Ç15
; L115
LOAD      F0009A
OUT       M1153F	// STEP Á¶°Ç16
// output comment: 04_ÀÚµ¿ STEP END
// ======================== ÀÛ¾÷ ¿Ï·á ==========================
; L117
LOAD      M11580	// L_TOOL CYCLE RUN
LOAD      M1151B	// 04_ Cycle end
OR        M1169F	// L_4th TOOL ÀÚÀç ¾ø¾îÁü
AND LOAD
OR        M11680	// L_4th TOOL ÀÛ¾÷¿Ï·á
AND       P00110	// L_4th DIE VACUUM EJECTOR ON
AND NOT   M11694	// L_4th TOOL ÀÚÀç °¡Á®°¨
OUT       M11680	// L_4th TOOL ÀÛ¾÷¿Ï·á

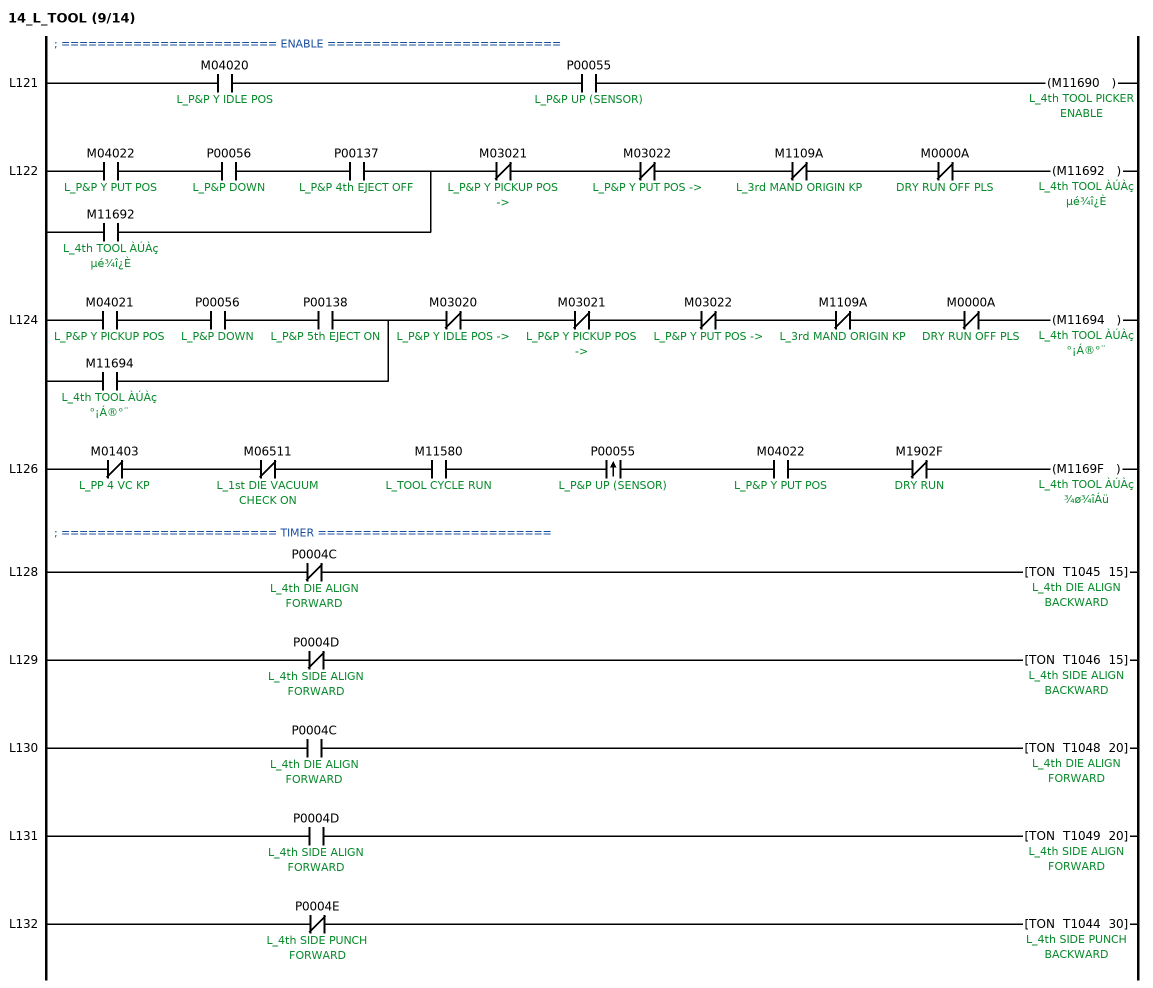
// ======================== ENABLE ==========================
; L121
LOAD      M04020	// L_P&P Y IDLE POS
AND       P00055	// L_P&P UP (SENSOR)
OUT       M11690	// L_4th TOOL PICKER ENABLE
; L122
LOAD      M04022	// L_P&P Y PUT POS
AND       P00056	// L_P&P DOWN
AND       P00137	// L_P&P 4th EJECT OFF
OR        M11692	// L_4th TOOL ÀÚÀç µé¾î¿È
AND NOT   M03021	// L_P&P Y PICKUP POS ->
AND NOT   M03022	// L_P&P Y PUT POS ->
AND NOT   M1109A	// L_3rd MAND ORIGIN KP
AND NOT   M0000A	// DRY RUN OFF PLS
OUT       M11692	// L_4th TOOL ÀÚÀç µé¾î¿È
; L124
LOAD      M04021	// L_P&P Y PICKUP POS
AND       P00056	// L_P&P DOWN
AND       P00138	// L_P&P 5th EJECT ON
OR        M11694	// L_4th TOOL ÀÚÀç °¡Á®°¨
AND NOT   M03020	// L_P&P Y IDLE POS ->
AND NOT   M03021	// L_P&P Y PICKUP POS ->
AND NOT   M03022	// L_P&P Y PUT POS ->
AND NOT   M1109A	// L_3rd MAND ORIGIN KP
AND NOT   M0000A	// DRY RUN OFF PLS
OUT       M11694	// L_4th TOOL ÀÚÀç °¡Á®°¨
; L126
LOAD NOT  M01403	// L_PP 4 VC KP
AND NOT   M06511	// L_1st DIE VACUUM CHECK ON
AND       M11580	// L_TOOL CYCLE RUN
ANDP      P00055	// L_P&P UP (SENSOR)
AND       M04022	// L_P&P Y PUT POS
AND NOT   M1902F	// DRY RUN
OUT       M1169F	// L_4th TOOL ÀÚÀç ¾ø¾îÁü
// ======================== TIMER ==========================
; L128
LOAD NOT  P0004C	// L_4th DIE ALIGN FORWARD
TON       T1045 15	// L_4th DIE ALIGN BACKWARD
; L129
LOAD NOT  P0004D	// L_4th SIDE ALIGN FORWARD
TON       T1046 15	// L_4th SIDE ALIGN BACKWARD
; L130
LOAD      P0004C	// L_4th DIE ALIGN FORWARD
TON       T1048 20	// L_4th DIE ALIGN FORWARD
; L131
LOAD      P0004D	// L_4th SIDE ALIGN FORWARD
TON       T1049 20	// L_4th SIDE ALIGN FORWARD
; L132
LOAD NOT  P0004E	// L_4th SIDE PUNCH FORWARD
TON       T1044 30	// L_4th SIDE PUNCH BACKWARD

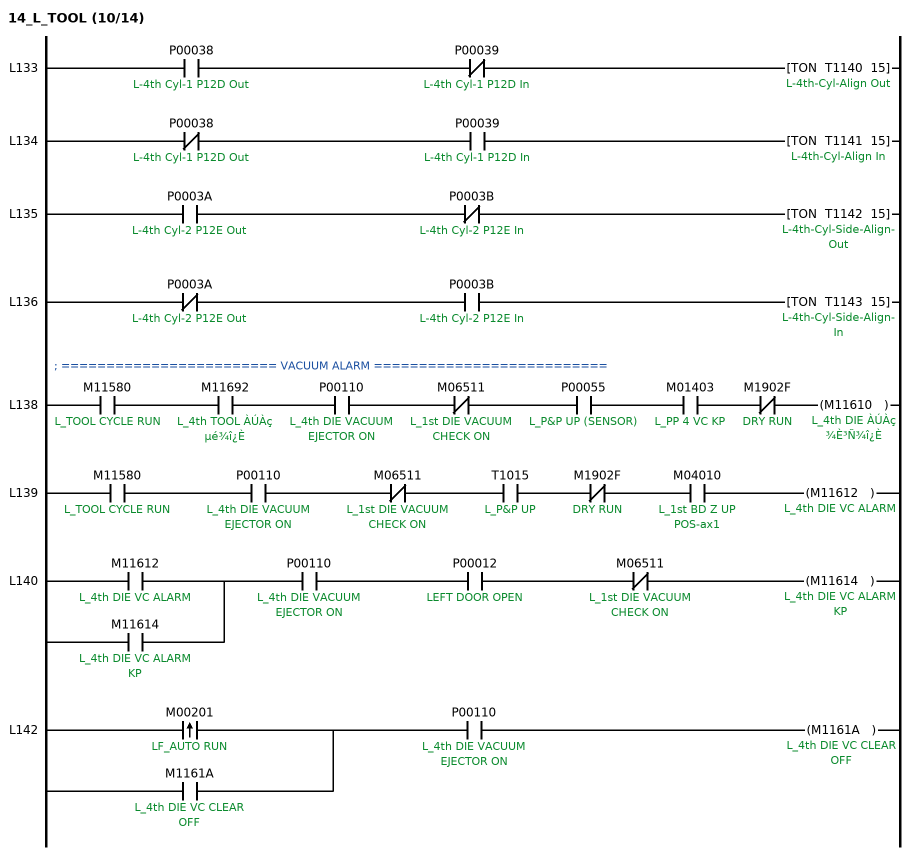
; L133
LOAD      P00038	// L-4th Cyl-1 P12D Out
AND NOT   P00039	// L-4th Cyl-1 P12D In
TON       T1140 15	// L-4th-Cyl-Align Out
; L134
LOAD NOT  P00038	// L-4th Cyl-1 P12D Out
AND       P00039	// L-4th Cyl-1 P12D In
TON       T1141 15	// L-4th-Cyl-Align In
; L135
LOAD      P0003A	// L-4th Cyl-2 P12E Out
AND NOT   P0003B	// L-4th Cyl-2 P12E In
TON       T1142 15	// L-4th-Cyl-Side-Align-Out
; L136
LOAD NOT  P0003A	// L-4th Cyl-2 P12E Out
AND       P0003B	// L-4th Cyl-2 P12E In
TON       T1143 15	// L-4th-Cyl-Side-Align-In
// ======================== VACUUM ALARM ==========================
; L138
LOAD      M11580	// L_TOOL CYCLE RUN
AND       M11692	// L_4th TOOL ÀÚÀç µé¾î¿È
AND       P00110	// L_4th DIE VACUUM EJECTOR ON
AND NOT   M06511	// L_1st DIE VACUUM CHECK ON
AND       P00055	// L_P&P UP (SENSOR)
AND       M01403	// L_PP 4 VC KP
AND NOT   M1902F	// DRY RUN
OUT       M11610	// L_4th DIE ÀÚÀç ¾È³Ñ¾î¿È
; L139
LOAD      M11580	// L_TOOL CYCLE RUN
AND       P00110	// L_4th DIE VACUUM EJECTOR ON
AND NOT   M06511	// L_1st DIE VACUUM CHECK ON
AND       T1015	// L_P&P UP
AND NOT   M1902F	// DRY RUN
AND       M04010	// L_1st BD Z UP POS-ax1
OUT       M11612	// L_4th DIE VC ALARM
; L140
LOAD      M11612	// L_4th DIE VC ALARM
OR        M11614	// L_4th DIE VC ALARM KP
AND       P00110	// L_4th DIE VACUUM EJECTOR ON
AND       P00012	// LEFT DOOR OPEN
AND NOT   M06511	// L_1st DIE VACUUM CHECK ON
OUT       M11614	// L_4th DIE VC ALARM KP
; L142
LOADP     M00201	// LF_AUTO RUN
OR        M1161A	// L_4th DIE VC CLEAR OFF
AND       P00110	// L_4th DIE VACUUM EJECTOR ON
OUT       M1161A	// L_4th DIE VC CLEAR OFF

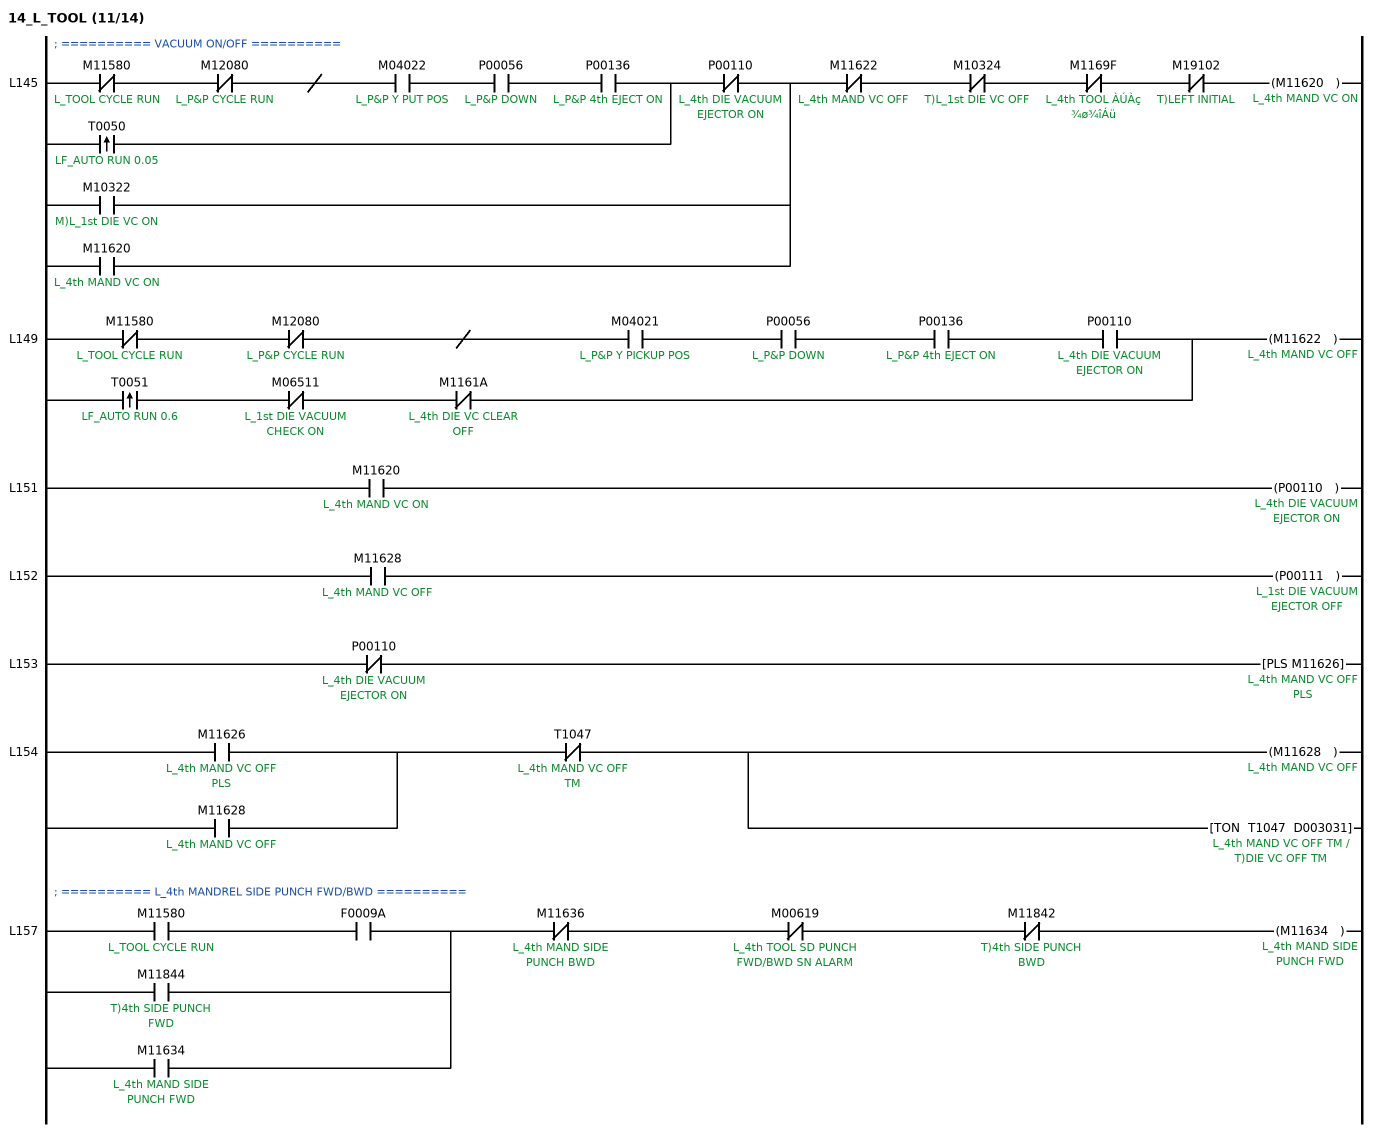
// ========== VACUUM ON/OFF ==========
; L145
LOAD NOT  M11580	// L_TOOL CYCLE RUN
AND NOT   M12080	// L_P&P CYCLE RUN
NOT
AND       M04022	// L_P&P Y PUT POS
AND       P00056	// L_P&P DOWN
AND       P00136	// L_P&P 4th EJECT ON
ORP       T0050	// LF_AUTO RUN 0.05
AND NOT   P00110	// L_4th DIE VACUUM EJECTOR ON
OR        M10322	// M)L_1st DIE VC ON
OR        M11620	// L_4th MAND VC ON
AND NOT   M11622	// L_4th MAND VC OFF
AND NOT   M10324	// T)L_1st DIE VC OFF
AND NOT   M1169F	// L_4th TOOL ÀÚÀç ¾ø¾îÁü
AND NOT   M19102	// T)LEFT INITIAL
OUT       M11620	// L_4th MAND VC ON
; L149
LOAD NOT  M11580	// L_TOOL CYCLE RUN
AND NOT   M12080	// L_P&P CYCLE RUN
NOT
AND       M04021	// L_P&P Y PICKUP POS
AND       P00056	// L_P&P DOWN
AND       P00136	// L_P&P 4th EJECT ON
AND       P00110	// L_4th DIE VACUUM EJECTOR ON
LOADP     T0051	// LF_AUTO RUN 0.6
AND NOT   M06511	// L_1st DIE VACUUM CHECK ON
AND NOT   M1161A	// L_4th DIE VC CLEAR OFF
OR LOAD
OUT       M11622	// L_4th MAND VC OFF
; L151
LOAD      M11620	// L_4th MAND VC ON
OUT       P00110	// L_4th DIE VACUUM EJECTOR ON
; L152
LOAD      M11628	// L_4th MAND VC OFF
OUT       P00111	// L_1st DIE VACUUM EJECTOR OFF
; L153
LOAD NOT  P00110	// L_4th DIE VACUUM EJECTOR ON
OUTP      M11626	// L_4th MAND VC OFF PLS
; L154
LOAD      M11626	// L_4th MAND VC OFF PLS
OR        M11628	// L_4th MAND VC OFF
AND NOT   T1047	// L_4th MAND VC OFF TM
OUT       M11628	// L_4th MAND VC OFF
TON       T1047 D003031	// L_4th MAND VC OFF TM / T)DIE VC OFF TM
// ========== L_4th MANDREL SIDE PUNCH FWD/BWD ==========
; L157
LOAD      M11580	// L_TOOL CYCLE RUN
AND       F0009A
OR        M11844	// T)4th SIDE PUNCH FWD
OR        M11634	// L_4th MAND SIDE PUNCH FWD
AND NOT   M11636	// L_4th MAND SIDE PUNCH BWD
AND NOT   M00619	// L_4th TOOL SD PUNCH FWD/BWD SN ALARM
AND NOT   M11842	// T)4th SIDE PUNCH BWD
OUT       M11634	// L_4th MAND SIDE PUNCH FWD

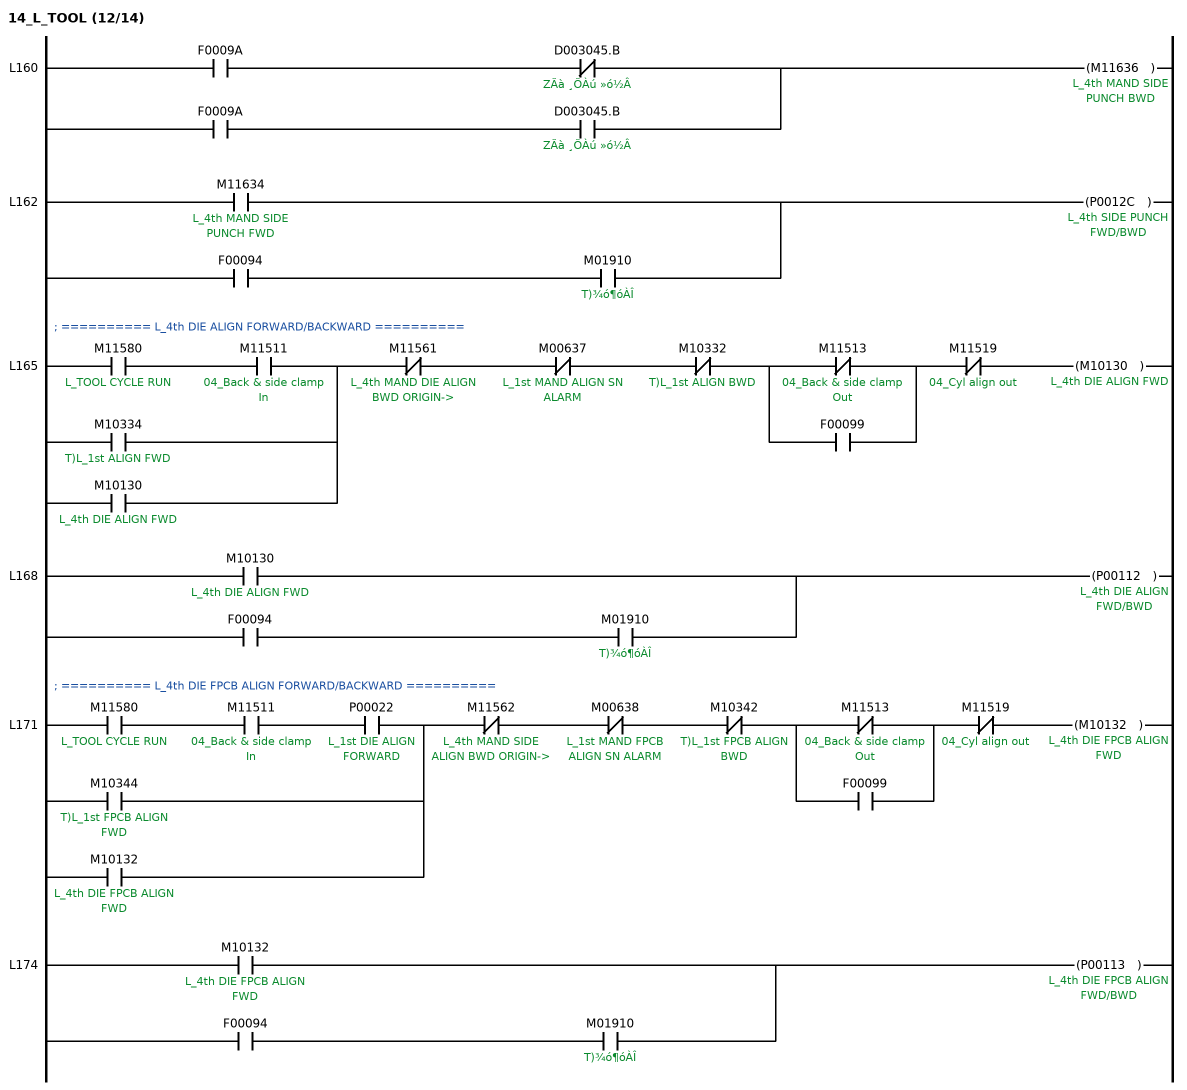
; L160
LOAD      F0009A
AND NOT   D003045.B	// ZÃà ¸ÕÀú »ó½Â
LOAD      F0009A
AND       D003045.B	// ZÃà ¸ÕÀú »ó½Â
OR LOAD
OUT       M11636	// L_4th MAND SIDE PUNCH BWD
; L162
LOAD      M11634	// L_4th MAND SIDE PUNCH FWD
LOAD      F00094
AND       M01910	// T)¾ó¶óÀÎ
OR LOAD
OUT       P0012C	// L_4th SIDE PUNCH FWD/BWD
// ========== L_4th DIE ALIGN FORWARD/BACKWARD ==========
; L165
LOAD      M11580	// L_TOOL CYCLE RUN
AND       M11511	// 04_Back & side clamp In
OR        M10334	// T)L_1st ALIGN FWD
OR        M10130	// L_4th DIE ALIGN FWD
AND NOT   M11561	// L_4th MAND DIE ALIGN BWD ORIGIN->
AND NOT   M00637	// L_1st MAND ALIGN SN ALARM
AND NOT   M10332	// T)L_1st ALIGN BWD
LOAD NOT  M11513	// 04_Back & side clamp Out
OR        F00099
AND LOAD
AND NOT   M11519	// 04_Cyl align out
OUT       M10130	// L_4th DIE ALIGN FWD
; L168
LOAD      M10130	// L_4th DIE ALIGN FWD
LOAD      F00094
AND       M01910	// T)¾ó¶óÀÎ
OR LOAD
OUT       P00112	// L_4th DIE ALIGN FWD/BWD
// ========== L_4th DIE FPCB ALIGN FORWARD/BACKWARD ==========
; L171
LOAD      M11580	// L_TOOL CYCLE RUN
AND       M11511	// 04_Back & side clamp In
AND       P00022	// L_1st DIE ALIGN FORWARD
OR        M10344	// T)L_1st FPCB ALIGN FWD
OR        M10132	// L_4th DIE FPCB ALIGN FWD
AND NOT   M11562	// L_4th MAND SIDE ALIGN BWD ORIGIN->
AND NOT   M00638	// L_1st MAND FPCB ALIGN SN ALARM
AND NOT   M10342	// T)L_1st FPCB ALIGN BWD
LOAD NOT  M11513	// 04_Back & side clamp Out
OR        F00099
AND LOAD
AND NOT   M11519	// 04_Cyl align out
OUT       M10132	// L_4th DIE FPCB ALIGN FWD
; L174
LOAD      M10132	// L_4th DIE FPCB ALIGN FWD
LOAD      F00094
AND       M01910	// T)¾ó¶óÀÎ
OR LOAD
OUT       P00113	// L_4th DIE FPCB ALIGN FWD/BWD

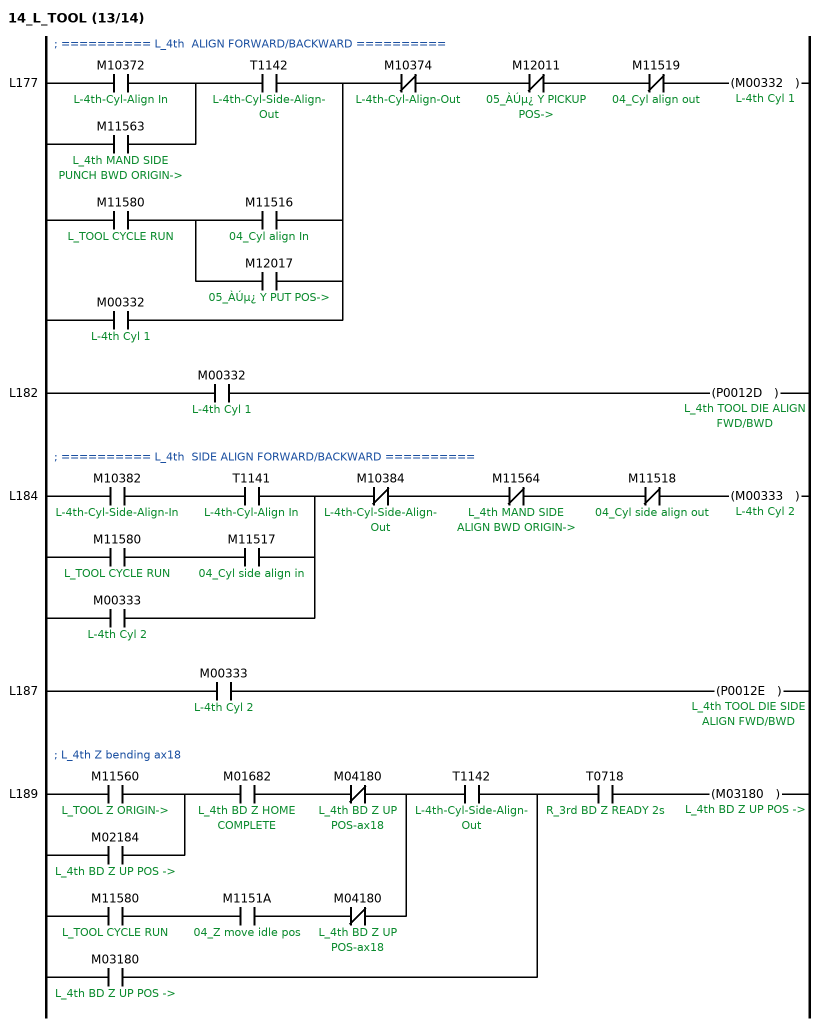
// ========== L_4th  ALIGN FORWARD/BACKWARD ==========
; L177
LOAD      M10372	// L-4th-Cyl-Align In
OR        M11563	// L_4th MAND SIDE PUNCH BWD ORIGIN->
AND       T1142	// L-4th-Cyl-Side-Align-Out
LOAD      M11580	// L_TOOL CYCLE RUN
LOAD      M11516	// 04_Cyl align In
OR        M12017	// 05_ÀÚµ¿ Y PUT POS->
AND LOAD
OR LOAD
OR        M00332	// L-4th Cyl 1
AND NOT   M10374	// L-4th-Cyl-Align-Out
AND NOT   M12011	// 05_ÀÚµ¿ Y PICKUP POS->
AND NOT   M11519	// 04_Cyl align out
OUT       M00332	// L-4th Cyl 1
; L182
LOAD      M00332	// L-4th Cyl 1
OUT       P0012D	// L_4th TOOL DIE ALIGN FWD/BWD
// ========== L_4th  SIDE ALIGN FORWARD/BACKWARD ==========
; L184
LOAD      M10382	// L-4th-Cyl-Side-Align-In
AND       T1141	// L-4th-Cyl-Align In
LOAD      M11580	// L_TOOL CYCLE RUN
AND       M11517	// 04_Cyl side align in
OR LOAD
OR        M00333	// L-4th Cyl 2
AND NOT   M10384	// L-4th-Cyl-Side-Align-Out
AND NOT   M11564	// L_4th MAND SIDE ALIGN BWD ORIGIN->
AND NOT   M11518	// 04_Cyl side align out
OUT       M00333	// L-4th Cyl 2
; L187
LOAD      M00333	// L-4th Cyl 2
OUT       P0012E	// L_4th TOOL DIE SIDE ALIGN FWD/BWD
// L_4th Z bending ax18
; L189
LOAD      M11560	// L_TOOL Z ORIGIN->
OR        M02184	// L_4th BD Z UP POS ->
AND       M01682	// L_4th BD Z HOME COMPLETE
AND NOT   M04180	// L_4th BD Z UP POS-ax18
LOAD      M11580	// L_TOOL CYCLE RUN
AND       M1151A	// 04_Z move idle pos
AND NOT   M04180	// L_4th BD Z UP POS-ax18
OR LOAD
AND       T1142	// L-4th-Cyl-Side-Align-Out
OR        M03180	// L_4th BD Z UP POS ->
AND       T0718	// R_3rd BD Z READY 2s
OUT       M03180	// L_4th BD Z UP POS ->

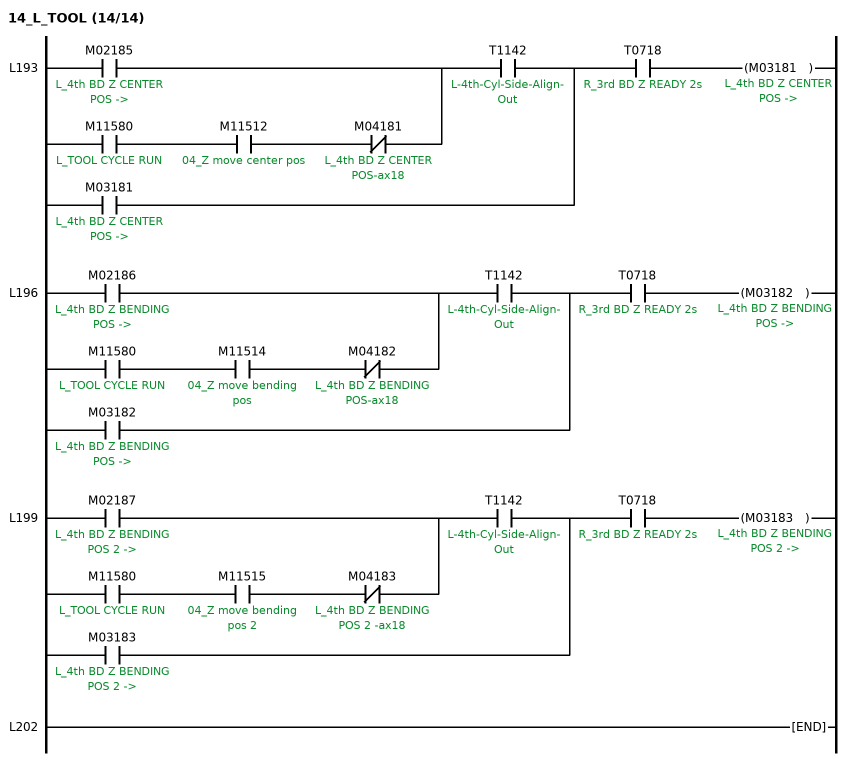
; L193
LOAD      M02185	// L_4th BD Z CENTER POS ->
LOAD      M11580	// L_TOOL CYCLE RUN
AND       M11512	// 04_Z move center pos
AND NOT   M04181	// L_4th BD Z CENTER POS-ax18
OR LOAD
AND       T1142	// L-4th-Cyl-Side-Align-Out
OR        M03181	// L_4th BD Z CENTER POS ->
AND       T0718	// R_3rd BD Z READY 2s
OUT       M03181	// L_4th BD Z CENTER POS ->
; L196
LOAD      M02186	// L_4th BD Z BENDING POS ->
LOAD      M11580	// L_TOOL CYCLE RUN
AND       M11514	// 04_Z move bending pos
AND NOT   M04182	// L_4th BD Z BENDING POS-ax18
OR LOAD
AND       T1142	// L-4th-Cyl-Side-Align-Out
OR        M03182	// L_4th BD Z BENDING POS ->
AND       T0718	// R_3rd BD Z READY 2s
OUT       M03182	// L_4th BD Z BENDING POS ->
; L199
LOAD      M02187	// L_4th BD Z BENDING POS 2 ->
LOAD      M11580	// L_TOOL CYCLE RUN
AND       M11515	// 04_Z move bending pos 2
AND NOT   M04183	// L_4th BD Z BENDING POS 2 -ax18
OR LOAD
AND       T1142	// L-4th-Cyl-Side-Align-Out
OR        M03183	// L_4th BD Z BENDING POS 2 ->
AND       T0718	// R_3rd BD Z READY 2s
OUT       M03183	// L_4th BD Z BENDING POS 2 ->
; L202
END

PROGRAM 15_L_PP (task: ½ºÄµ ÇÁ·Î±×·¥)

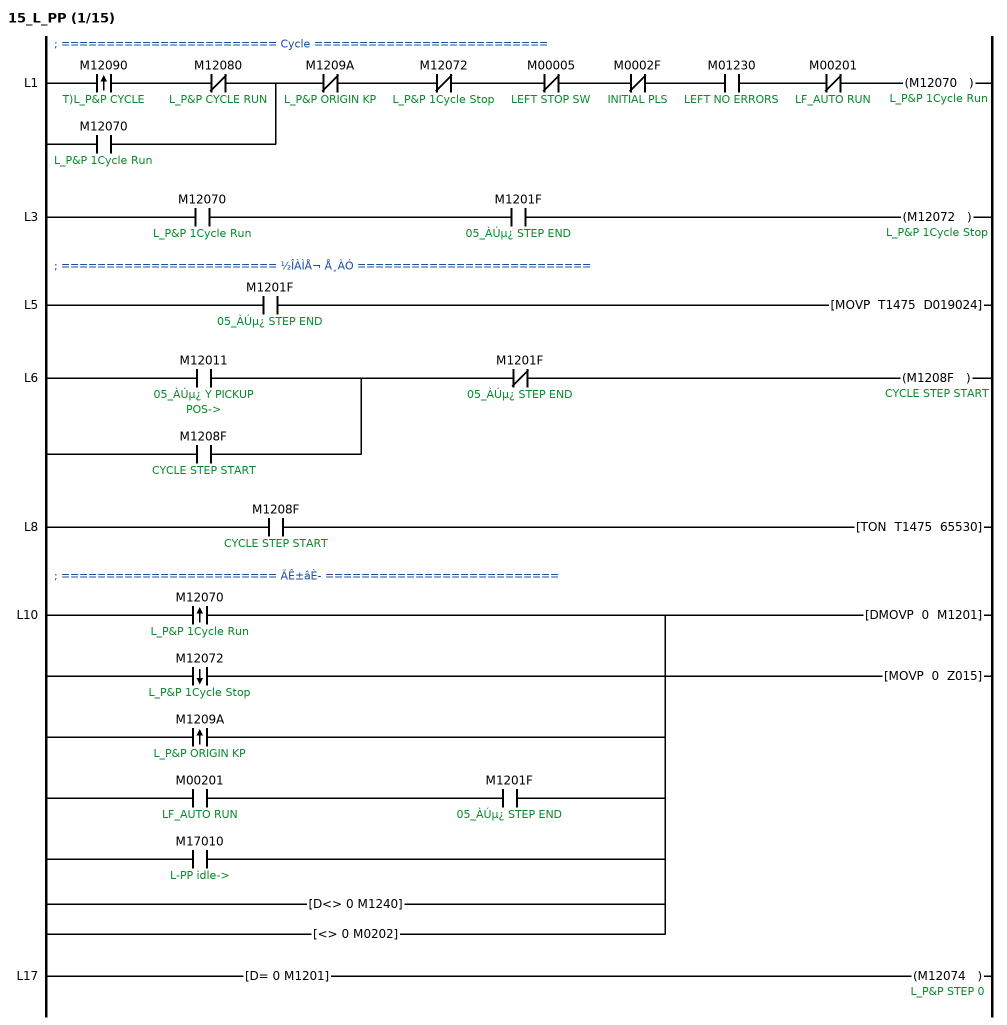
// ======================== Cycle ==========================
; L1
LOADP     M12090	// T)L_P&P CYCLE
AND NOT   M12080	// L_P&P CYCLE RUN
OR        M12070	// L_P&P 1Cycle Run
AND NOT   M1209A	// L_P&P ORIGIN KP
AND NOT   M12072	// L_P&P 1Cycle Stop
AND NOT   M00005	// LEFT STOP SW
AND NOT   M0002F	// INITIAL PLS
AND       M01230	// LEFT NO ERRORS
AND NOT   M00201	// LF_AUTO RUN
OUT       M12070	// L_P&P 1Cycle Run
; L3
LOAD      M12070	// L_P&P 1Cycle Run
AND       M1201F	// 05_ÀÚµ¿ STEP END
OUT       M12072	// L_P&P 1Cycle Stop
// ======================== ½ÎÀÌÅ¬ Å¸ÀÓ ==========================
; L5
LOAD      M1201F	// 05_ÀÚµ¿ STEP END
MOVP      T1475 D019024
; L6
LOAD      M12011	// 05_ÀÚµ¿ Y PICKUP POS->
OR        M1208F	// CYCLE STEP START
AND NOT   M1201F	// 05_ÀÚµ¿ STEP END
OUT       M1208F	// CYCLE STEP START
; L8
LOAD      M1208F	// CYCLE STEP START
TON       T1475 65530
// ======================== ÃÊ±âÈ­ ==========================
; L10
LOADP     M12070	// L_P&P 1Cycle Run
ORN       M12072	// L_P&P 1Cycle Stop
ORP       M1209A	// L_P&P ORIGIN KP
LOAD      M00201	// LF_AUTO RUN
AND       M1201F	// 05_ÀÚµ¿ STEP END
OR LOAD
OR        M17010	// L-PP idle->
ORD<>     0 M1240
OR<>      0 M0202
DMOVP     0 M1201
MOVP      0 Z015
; L17
LOADD=    0 M1201
OUT       M12074	// L_P&P STEP 0

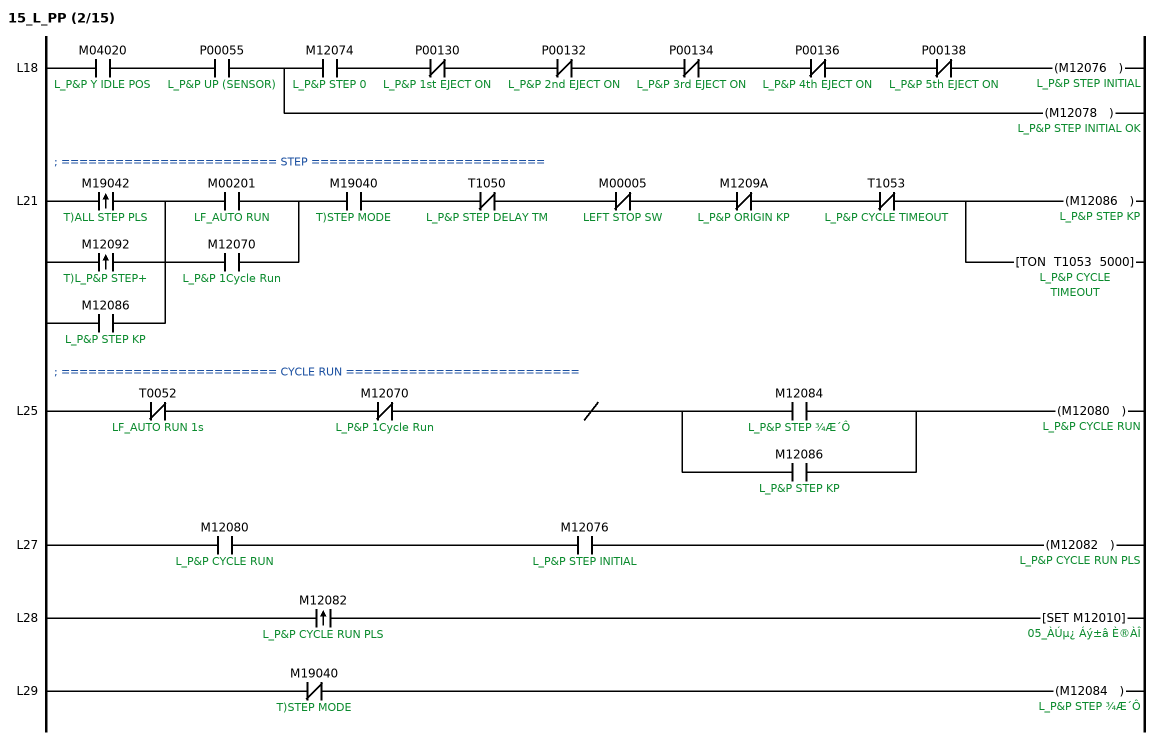
; L18
LOAD      M04020	// L_P&P Y IDLE POS
AND       P00055	// L_P&P UP (SENSOR)
MPUSH
AND       M12074	// L_P&P STEP 0
AND NOT   P00130	// L_P&P 1st EJECT ON
AND NOT   P00132	// L_P&P 2nd EJECT ON
AND NOT   P00134	// L_P&P 3rd EJECT ON
AND NOT   P00136	// L_P&P 4th EJECT ON
AND NOT   P00138	// L_P&P 5th EJECT ON
OUT       M12076	// L_P&P STEP INITIAL
MPOP
OUT       M12078	// L_P&P STEP INITIAL OK
// ======================== STEP ==========================
; L21
LOADP     M19042	// T)ALL STEP PLS
ORP       M12092	// T)L_P&P STEP+
OR        M12086	// L_P&P STEP KP
LOAD      M00201	// LF_AUTO RUN
OR        M12070	// L_P&P 1Cycle Run
AND LOAD
AND       M19040	// T)STEP MODE
AND NOT   T1050	// L_P&P STEP DELAY TM
AND NOT   M00005	// LEFT STOP SW
AND NOT   M1209A	// L_P&P ORIGIN KP
AND NOT   T1053	// L_P&P CYCLE TIMEOUT
OUT       M12086	// L_P&P STEP KP
TON       T1053 5000	// L_P&P CYCLE TIMEOUT
// ======================== CYCLE RUN ==========================
; L25
LOAD NOT  T0052	// LF_AUTO RUN 1s
AND NOT   M12070	// L_P&P 1Cycle Run
NOT
LOAD      M12084	// L_P&P STEP ¾Æ´Ô
OR        M12086	// L_P&P STEP KP
AND LOAD
OUT       M12080	// L_P&P CYCLE RUN
; L27
LOAD      M12080	// L_P&P CYCLE RUN
AND       M12076	// L_P&P STEP INITIAL
OUT       M12082	// L_P&P CYCLE RUN PLS
; L28
LOADP     M12082	// L_P&P CYCLE RUN PLS
SET       M12010	// 05_ÀÚµ¿ Áý±â È®ÀÎ
; L29
LOAD NOT  M19040	// T)STEP MODE
OUT       M12084	// L_P&P STEP ¾Æ´Ô

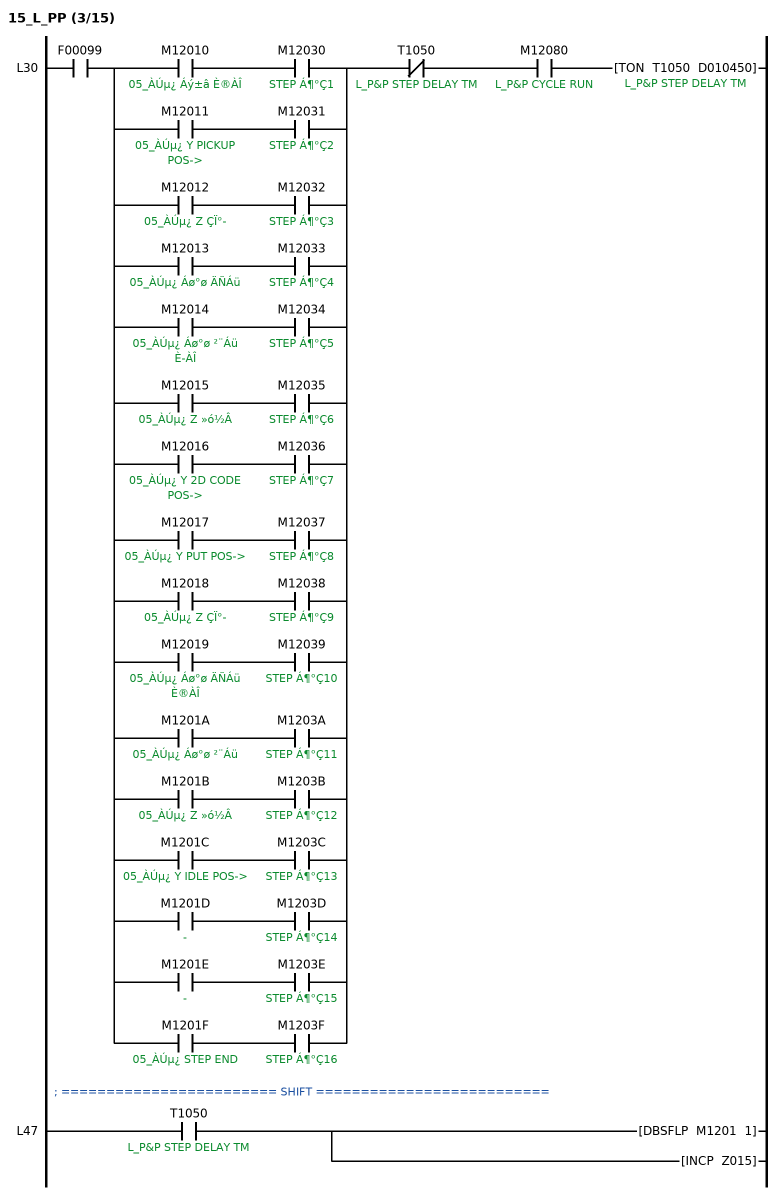
; L30
LOAD      F00099
LOAD      M12010	// 05_ÀÚµ¿ Áý±â È®ÀÎ
AND       M12030	// STEP Á¶°Ç1
LOAD      M12011	// 05_ÀÚµ¿ Y PICKUP POS->
AND       M12031	// STEP Á¶°Ç2
OR LOAD
LOAD      M12012	// 05_ÀÚµ¿ Z ÇÏ°­
AND       M12032	// STEP Á¶°Ç3
OR LOAD
LOAD      M12013	// 05_ÀÚµ¿ Áø°ø ÄÑÁü
AND       M12033	// STEP Á¶°Ç4
OR LOAD
LOAD      M12014	// 05_ÀÚµ¿ Áø°ø ²¨Áü È­ÀÎ
AND       M12034	// STEP Á¶°Ç5
OR LOAD
LOAD      M12015	// 05_ÀÚµ¿ Z »ó½Â
AND       M12035	// STEP Á¶°Ç6
OR LOAD
LOAD      M12016	// 05_ÀÚµ¿ Y 2D CODE POS->
AND       M12036	// STEP Á¶°Ç7
OR LOAD
LOAD      M12017	// 05_ÀÚµ¿ Y PUT POS->
AND       M12037	// STEP Á¶°Ç8
OR LOAD
LOAD      M12018	// 05_ÀÚµ¿ Z ÇÏ°­
AND       M12038	// STEP Á¶°Ç9
OR LOAD
LOAD      M12019	// 05_ÀÚµ¿ Áø°ø ÄÑÁü È®ÀÎ
AND       M12039	// STEP Á¶°Ç10
OR LOAD
LOAD      M1201A	// 05_ÀÚµ¿ Áø°ø ²¨Áü
AND       M1203A	// STEP Á¶°Ç11
OR LOAD
LOAD      M1201B	// 05_ÀÚµ¿ Z »ó½Â
AND       M1203B	// STEP Á¶°Ç12
OR LOAD
LOAD      M1201C	// 05_ÀÚµ¿ Y IDLE POS->
AND       M1203C	// STEP Á¶°Ç13
OR LOAD
LOAD      M1201D	// -
AND       M1203D	// STEP Á¶°Ç14
OR LOAD
LOAD      M1201E	// -
AND       M1203E	// STEP Á¶°Ç15
OR LOAD
LOAD      M1201F	// 05_ÀÚµ¿ STEP END
AND       M1203F	// STEP Á¶°Ç16
OR LOAD
AND LOAD
AND NOT   T1050	// L_P&P STEP DELAY TM
AND       M12080	// L_P&P CYCLE RUN
TON       T1050 D010450	// L_P&P STEP DELAY TM
// ======================== SHIFT ==========================
; L47
LOAD      T1050	// L_P&P STEP DELAY TM
DBSFLP    M1201 1
INCP      Z015

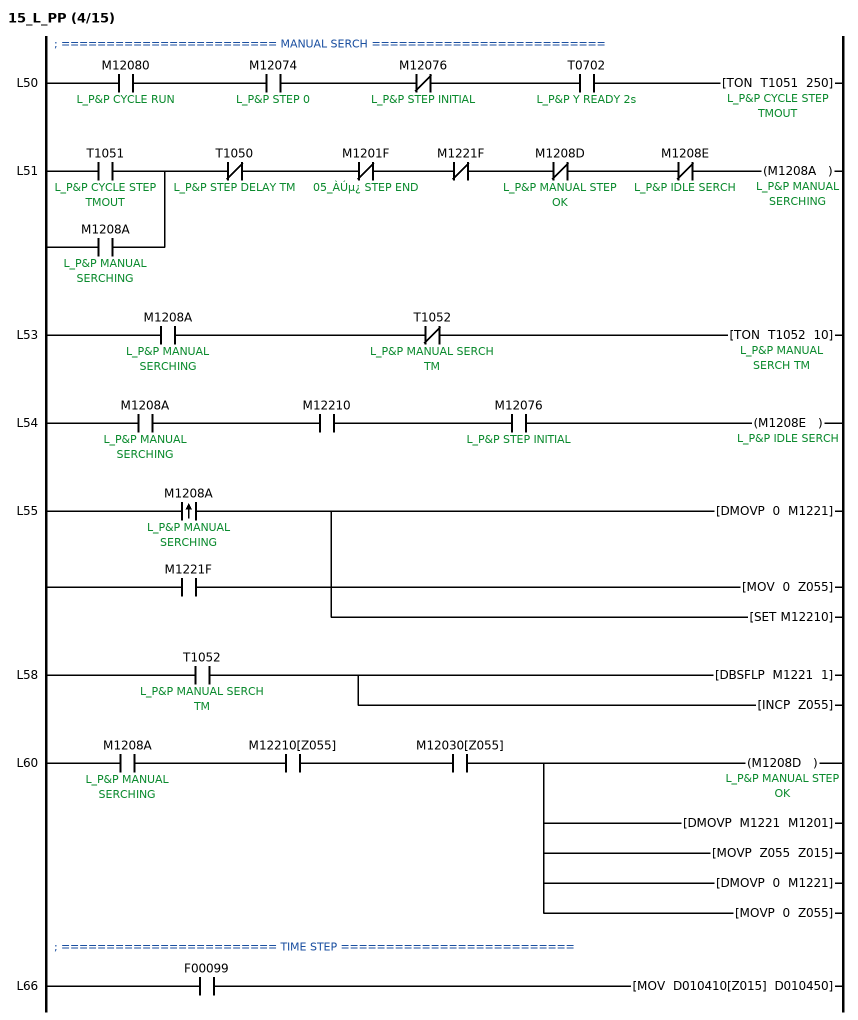
// ======================== MANUAL SERCH ==========================
; L50
LOAD      M12080	// L_P&P CYCLE RUN
AND       M12074	// L_P&P STEP 0
AND NOT   M12076	// L_P&P STEP INITIAL
AND       T0702	// L_P&P Y READY 2s
TON       T1051 250	// L_P&P CYCLE STEP TMOUT
; L51
LOAD      T1051	// L_P&P CYCLE STEP TMOUT
OR        M1208A	// L_P&P MANUAL SERCHING
AND NOT   T1050	// L_P&P STEP DELAY TM
AND NOT   M1201F	// 05_ÀÚµ¿ STEP END
AND NOT   M1221F
AND NOT   M1208D	// L_P&P MANUAL STEP OK
AND NOT   M1208E	// L_P&P IDLE SERCH
OUT       M1208A	// L_P&P MANUAL SERCHING
; L53
LOAD      M1208A	// L_P&P MANUAL SERCHING
AND NOT   T1052	// L_P&P MANUAL SERCH TM
TON       T1052 10	// L_P&P MANUAL SERCH TM
; L54
LOAD      M1208A	// L_P&P MANUAL SERCHING
AND       M12210
AND       M12076	// L_P&P STEP INITIAL
OUT       M1208E	// L_P&P IDLE SERCH
; L55
LOADP     M1208A	// L_P&P MANUAL SERCHING
OR        M1221F
DMOVP     0 M1221
MOV       0 Z055
SET       M12210
; L58
LOAD      T1052	// L_P&P MANUAL SERCH TM
DBSFLP    M1221 1
INCP      Z055
; L60
LOAD      M1208A	// L_P&P MANUAL SERCHING
AND       M12210[Z055]
AND       M12030[Z055]
OUT       M1208D	// L_P&P MANUAL STEP OK
DMOVP     M1221 M1201
MOVP      Z055 Z015
DMOVP     0 M1221
MOVP      0 Z055
// ======================== TIME STEP ==========================
; L66
LOAD      F00099
MOV       D010410[Z015] D010450

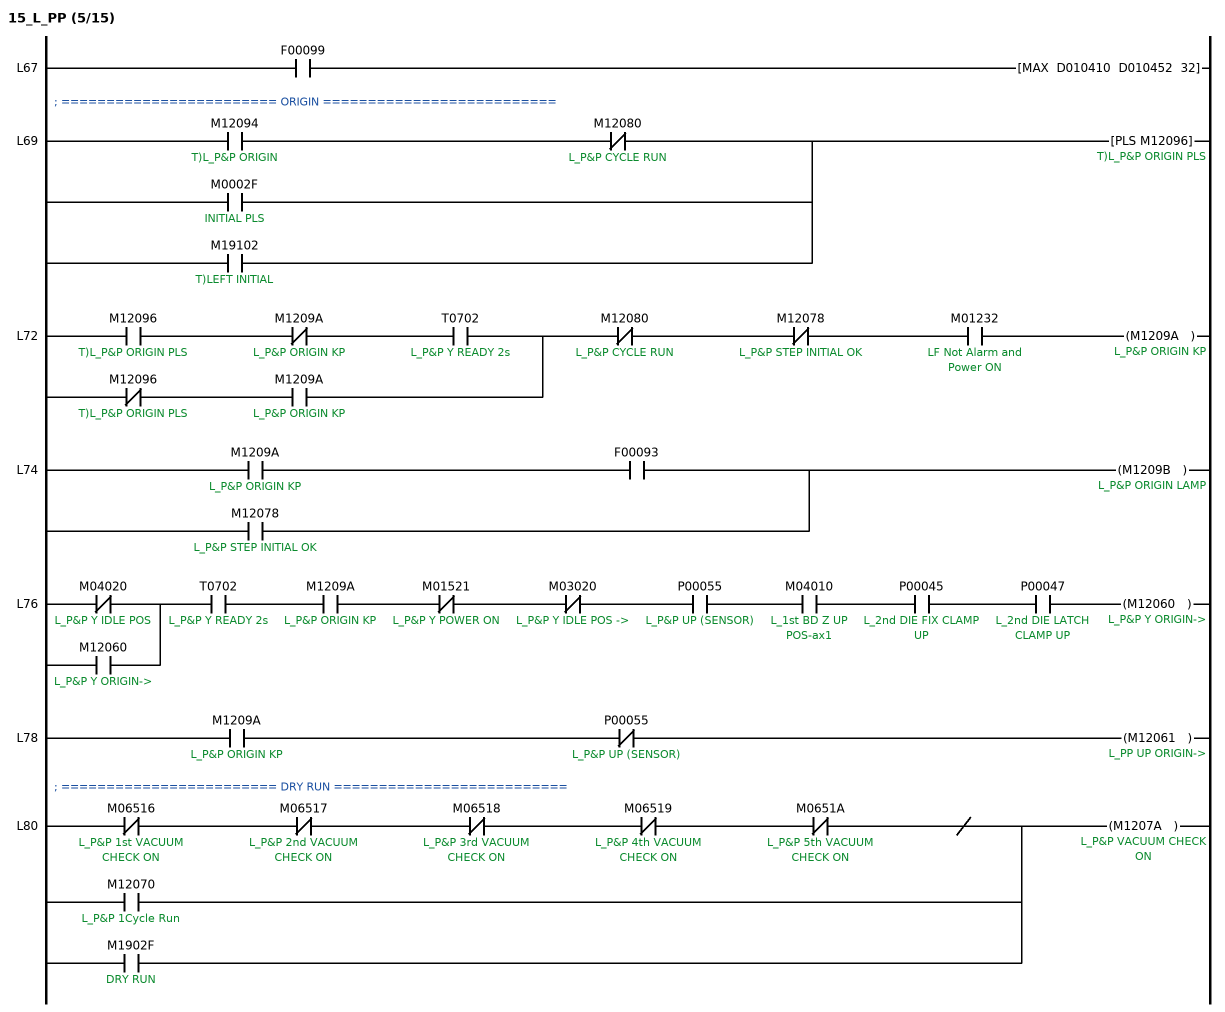
; L67
LOAD      F00099
MAX       D010410 D010452 32
// ======================== ORIGIN ==========================
; L69
LOAD      M12094	// T)L_P&P ORIGIN
AND NOT   M12080	// L_P&P CYCLE RUN
OR        M0002F	// INITIAL PLS
OR        M19102	// T)LEFT INITIAL
OUTP      M12096	// T)L_P&P ORIGIN PLS
; L72
LOAD      M12096	// T)L_P&P ORIGIN PLS
AND NOT   M1209A	// L_P&P ORIGIN KP
AND       T0702	// L_P&P Y READY 2s
LOAD NOT  M12096	// T)L_P&P ORIGIN PLS
AND       M1209A	// L_P&P ORIGIN KP
OR LOAD
AND NOT   M12080	// L_P&P CYCLE RUN
AND NOT   M12078	// L_P&P STEP INITIAL OK
AND       M01232	// LF Not Alarm and Power ON
OUT       M1209A	// L_P&P ORIGIN KP
; L74
LOAD      M1209A	// L_P&P ORIGIN KP
AND       F00093
OR        M12078	// L_P&P STEP INITIAL OK
OUT       M1209B	// L_P&P ORIGIN LAMP
; L76
LOAD NOT  M04020	// L_P&P Y IDLE POS
OR        M12060	// L_P&P Y ORIGIN->
AND       T0702	// L_P&P Y READY 2s
AND       M1209A	// L_P&P ORIGIN KP
AND NOT   M01521	// L_P&P Y POWER ON
AND NOT   M03020	// L_P&P Y IDLE POS ->
AND       P00055	// L_P&P UP (SENSOR)
AND       M04010	// L_1st BD Z UP POS-ax1
AND       P00045	// L_2nd DIE FIX CLAMP UP
AND       P00047	// L_2nd DIE LATCH CLAMP UP
OUT       M12060	// L_P&P Y ORIGIN->
; L78
LOAD      M1209A	// L_P&P ORIGIN KP
AND NOT   P00055	// L_P&P UP (SENSOR)
OUT       M12061	// L_PP UP ORIGIN->
// ======================== DRY RUN ==========================
; L80
LOAD NOT  M06516	// L_P&P 1st VACUUM CHECK ON
AND NOT   M06517	// L_P&P 2nd VACUUM CHECK ON
AND NOT   M06518	// L_P&P 3rd VACUUM CHECK ON
AND NOT   M06519	// L_P&P 4th VACUUM CHECK ON
AND NOT   M0651A	// L_P&P 5th VACUUM CHECK ON
NOT
OR        M12070	// L_P&P 1Cycle Run
OR        M1902F	// DRY RUN
OUT       M1207A	// L_P&P VACUUM CHECK ON

